LIN {X 0,Y 425.323,Z 412.747,A -85,B 0,C 180,E1 20527.293,E2 20527.293} C_VEL
LIN {X 0,Y 425.31,Z 412.73,A -85,B 0,C 180,E1 20523.37,E2 20523.37} C_VEL
LIN {X 0,Y 425.312,Z 412.748,A -85,B 0,C 180,E1 20519.596,E2 20519.596} C_VEL
LIN {X 0,Y 425.314,Z 412.756,A -85,B 0,C 180,E1 20515.686,E2 20515.686} C_VEL
LIN {X 0,Y 425.313,Z 412.739,A -85,B 0,C 180,E1 20511.785,E2 20511.785} C_VEL
LIN {X 0,Y 425.305,Z 412.739,A -85,B 0,C 180,E1 20507.923,E2 20507.923} C_VEL
LIN {X 0,Y 425.305,Z 412.745,A -85,B 0,C 180,E1 20504.035,E2 20504.035} C_VEL
LIN {X 0,Y 425.315,Z 412.752,A -85,B 0,C 180,E1 20500.213,E2 20500.213} C_VEL
LIN {X 0,Y 425.319,Z 412.753,A -85,B 0,C 180,E1 20496.445,E2 20496.445} C_VEL
LIN {X 0,Y 425.317,Z 412.751,A -85,B 0,C 180,E1 20492.564,E2 20492.564} C_VEL
LIN {X 0,Y 425.318,Z 412.746,A -85,B 0,C 180,E1 20488.699,E2 20488.699} C_VEL
LIN {X 0,Y 425.308,Z 412.744,A -85,B 0,C 180,E1 20484.833,E2 20484.833} C_VEL
LIN {X 0,Y 425.354,Z 413.101,A -85,B 0,C 180,E1 20483.004,E2 20483.004} C_VEL
LIN {X 0,Y 426.927,Z 416.653,A -85,B 0,C 180,E1 20482.32,E2 20482.32} C_VEL
LIN {X 0,Y 432.518,Z 427.517,A -85,B 0,C 180,E1 20480.338,E2 20480.338} C_VEL
LIN {X 0,Y 440.168,Z 443.004,A -85,B 0,C 180,E1 20477.75,E2 20477.75} C_VEL
LIN {X 0,Y 445.904,Z 455.372,A -85,B 0,C 180,E1 20475.919,E2 20475.919} C_VEL
LIN {X 0,Y 457.025,Z 473.943,A -85,B 0,C 180,E1 20474.241,E2 20474.241} C_VEL
LIN {X 0,Y 458.912,Z 489.017,A -85,B 0,C 180,E1 20473.725,E2 20473.725} C_VEL
LIN {X 0,Y 453.234,Z 708.899,A -85,B 0,C 180,E1 20469.92,E2 20469.92} C_VEL
LIN {X 0,Y 451.808,Z 759.725,A -85,B 0,C 180,E1 20469.018,E2 20469.018} C_VEL
LIN {X 0,Y 450.365,Z 781.628,A -85,B 0,C 180,E1 20468.419,E2 20468.419} C_VEL
LIN {X 0,Y 448.539,Z 802.923,A -85,B 0,C 180,E1 20467.608,E2 20467.608} C_VEL
LIN {X 0,Y 446.493,Z 822.784,A -85,B 0,C 180,E1 20466.642,E2 20466.642} C_VEL
LIN {X 0,Y 444.028,Z 843.126,A -85,B 0,C 180,E1 20465.399,E2 20465.399} C_VEL
LIN {X 0,Y 441.405,Z 862.685,A -85,B 0,C 180,E1 20463.945,E2 20463.945} C_VEL
LIN {X 0,Y 438.705,Z 881.613,A -85,B 0,C 180,E1 20462.27,E2 20462.27} C_VEL
LIN {X 0,Y 436.022,Z 899.637,A -85,B 0,C 180,E1 20460.376,E2 20460.376} C_VEL
LIN {X 0,Y 433.447,Z 916.409,A -85,B 0,C 180,E1 20458.299,E2 20458.299} C_VEL
LIN {X 0,Y 430.956,Z 933.189,A -85,B 0,C 180,E1 20455.863,E2 20455.863} C_VEL
LIN {X 0,Y 429.001,Z 947.176,A -85,B 0,C 180,E1 20453.489,E2 20453.489} C_VEL
LIN {X 0,Y 427.354,Z 959.751,A -85,B 0,C 180,E1 20450.978,E2 20450.978} C_VEL
LIN {X 0,Y 426.064,Z 971.018,A -85,B 0,C 180,E1 20448.331,E2 20448.331} C_VEL
LIN {X 0,Y 425.116,Z 980.962,A -85,B 0,C 180,E1 20445.555,E2 20445.555} C_VEL
LIN {X 0,Y 424.496,Z 988.98,A -85,B 0,C 180,E1 20442.794,E2 20442.794} C_VEL
LIN {X 0,Y 424.128,Z 995.597,A -85,B 0,C 180,E1 20439.912,E2 20439.912} C_VEL
LIN {X 0,Y 423.966,Z 1000.343,A -85,B 0,C 180,E1 20437.183,E2 20437.183} C_VEL
LIN {X 0,Y 423.919,Z 1003.442,A -85,B 0,C 180,E1 20434.467,E2 20434.467} C_VEL
LIN {X 0,Y 423.901,Z 1005.174,A -85,B 0,C 180,E1 20431.76,E2 20431.76} C_VEL
LIN {X 0,Y 423.901,Z 1005.321,A -85,B 0,C 180,E1 20429.057,E2 20429.057} C_VEL
LIN {X 0,Y 423.913,Z 1004.043,A -85,B 0,C 180,E1 20426.216,E2 20426.216} C_VEL
LIN {X 0,Y 423.96,Z 1001.217,A -85,B 0,C 180,E1 20423.503,E2 20423.503} C_VEL
LIN {X 0,Y 424.094,Z 996.661,A -85,B 0,C 180,E1 20420.641,E2 20420.641} C_VEL
LIN {X 0,Y 424.374,Z 991.039,A -85,B 0,C 180,E1 20418.037,E2 20418.037} C_VEL
LIN {X 0,Y 424.881,Z 983.447,A -85,B 0,C 180,E1 20415.28,E2 20415.28} C_VEL
LIN {X 0,Y 425.72,Z 974.127,A -85,B 0,C 180,E1 20412.508,E2 20412.508} C_VEL
LIN {X 0,Y 426.887,Z 963.337,A -85,B 0,C 180,E1 20409.864,E2 20409.864} C_VEL
LIN {X 0,Y 428.486,Z 950.359,A -85,B 0,C 180,E1 20407.178,E2 20407.178} C_VEL
LIN {X 0,Y 430.41,Z 936.295,A -85,B 0,C 180,E1 20404.699,E2 20404.699} C_VEL
LIN {X 0,Y 432.667,Z 920.798,A -85,B 0,C 180,E1 20402.368,E2 20402.368} C_VEL
LIN {X 0,Y 435.099,Z 904.208,A -85,B 0,C 180,E1 20400.244,E2 20400.244} C_VEL
LIN {X 0,Y 437.815,Z 885.884,A -85,B 0,C 180,E1 20398.242,E2 20398.242} C_VEL
LIN {X 0,Y 440.47,Z 867.438,A -85,B 0,C 180,E1 20396.527,E2 20396.527} C_VEL
LIN {X 0,Y 443.06,Z 848.116,A -85,B 0,C 180,E1 20395.031,E2 20395.031} C_VEL
LIN {X 0,Y 445.48,Z 828.163,A -85,B 0,C 180,E1 20393.747,E2 20393.747} C_VEL
LIN {X 0,Y 447.727,Z 807.657,A -85,B 0,C 180,E1 20392.674,E2 20392.674} C_VEL
LIN {X 0,Y 449.569,Z 787.136,A -85,B 0,C 180,E1 20391.839,E2 20391.839} C_VEL
LIN {X 0,Y 451.131,Z 764.896,A -85,B 0,C 180,E1 20391.175,E2 20391.175} C_VEL
LIN {X 0,Y 452.115,Z 740.735,A -85,B 0,C 180,E1 20390.686,E2 20390.686} C_VEL
LIN {X 0,Y 457.722,Z 517.41,A -85,B 0,C 180,E1 20386.836,E2 20386.836} C_VEL
LIN {X 0,Y 458.387,Z 486.605,A -85,B 0,C 180,E1 20386.272,E2 20386.272} C_VEL
LIN {X 0,Y 456.382,Z 472.949,A -85,B 0,C 180,E1 20385.758,E2 20385.758} C_VEL
LIN {X 0,Y 445.388,Z 454.22,A -85,B 0,C 180,E1 20384.011,E2 20384.011} C_VEL
LIN {X 0,Y 438.051,Z 438.21,A -85,B 0,C 180,E1 20381.447,E2 20381.447} C_VEL
LIN {X 0,Y 431.895,Z 425.933,A -85,B 0,C 180,E1 20379.198,E2 20379.198} C_VEL
LIN {X 0,Y 429.067,Z 420.711,A -85,B 0,C 180,E1 20378.136,E2 20378.136} C_VEL
LIN {X 0,Y 427.444,Z 417.332,A -85,B 0,C 180,E1 20377.458,E2 20377.458} C_VEL
LIN {X 0,Y 425.676,Z 414.437,A -85,B 0,C 180,E1 20376.785,E2 20376.785} C_VEL
LIN {X 0,Y 425.321,Z 412.922,A -85,B 0,C 180,E1 20376.4,E2 20376.4} C_VEL
LIN {X 0,Y 425.274,Z 412.761,A -85,B 0,C 180,E1 20372.689,E2 20372.689} C_VEL
LIN {X 0,Y 425.267,Z 412.756,A -85,B 0,C 180,E1 20368.968,E2 20368.968} C_VEL
LIN {X 0,Y 425.272,Z 412.763,A -85,B 0,C 180,E1 20365.185,E2 20365.185} C_VEL
LIN {X 0,Y 425.292,Z 412.751,A -85,B 0,C 180,E1 20361.422,E2 20361.422} C_VEL
LIN {X 0,Y 425.293,Z 412.749,A -85,B 0,C 180,E1 20357.654,E2 20357.654} C_VEL
LIN {X 0,Y 425.262,Z 412.756,A -85,B 0,C 180,E1 20353.875,E2 20353.875} C_VEL
LIN {X 0,Y 425.248,Z 412.764,A -85,B 0,C 180,E1 20350.156,E2 20350.156} C_VEL
LIN {X 0,Y 425.253,Z 412.763,A -85,B 0,C 180,E1 20346.344,E2 20346.344} C_VEL
LIN {X 0,Y 425.267,Z 412.754,A -85,B 0,C 180,E1 20342.56,E2 20342.56} C_VEL
LIN {X 0,Y 425.307,Z 412.749,A -85,B 0,C 180,E1 20338.922,E2 20338.922} C_VEL
LIN {X 0,Y 425.316,Z 412.758,A -85,B 0,C 180,E1 20335.01,E2 20335.01} C_VEL
LIN {X 0,Y 425.309,Z 412.75,A -85,B 0,C 180,E1 20331.21,E2 20331.21} C_VEL
LIN {X 0,Y 425.298,Z 412.76,A -85,B 0,C 180,E1 20327.37,E2 20327.37} C_VEL
LIN {X 0,Y 425.335,Z 413.097,A -85,B 0,C 180,E1 20325.767,E2 20325.767} C_VEL
LIN {X 0,Y 426.924,Z 416.643,A -85,B 0,C 180,E1 20324.932,E2 20324.932} C_VEL
LIN {X 0,Y 428.049,Z 418.942,A -85,B 0,C 180,E1 20324.417,E2 20324.417} C_VEL
LIN {X 0,Y 431.92,Z 426.469,A -85,B 0,C 180,E1 20322.764,E2 20322.764} C_VEL
LIN {X 0,Y 438.754,Z 441.345,A -85,B 0,C 180,E1 20319.872,E2 20319.872} C_VEL
LIN {X 0,Y 443.854,Z 453.504,A -85,B 0,C 180,E1 20317.803,E2 20317.803} C_VEL
LIN {X 0,Y 453.373,Z 469.49,A -85,B 0,C 180,E1 20316.249,E2 20316.249} C_VEL
LIN {X 0,Y 455.989,Z 486.254,A -85,B 0,C 180,E1 20315.571,E2 20315.571} C_VEL
LIN {X 0,Y 448.514,Z 720.49,A -85,B 0,C 180,E1 20311.323,E2 20311.323} C_VEL
LIN {X 0,Y 447.258,Z 741.418,A -85,B 0,C 180,E1 20310.709,E2 20310.709} C_VEL
LIN {X 0,Y 445.663,Z 761.022,A -85,B 0,C 180,E1 20309.905,E2 20309.905} C_VEL
LIN {X 0,Y 443.641,Z 781.159,A -85,B 0,C 180,E1 20308.827,E2 20308.827} C_VEL
LIN {X 0,Y 441.338,Z 800.443,A -85,B 0,C 180,E1 20307.525,E2 20307.525} C_VEL
LIN {X 0,Y 439.005,Z 817.909,A -85,B 0,C 180,E1 20306.082,E2 20306.082} C_VEL
LIN {X 0,Y 436.526,Z 834.898,A -85,B 0,C 180,E1 20304.395,E2 20304.395} C_VEL
LIN {X 0,Y 434.09,Z 850.626,A -85,B 0,C 180,E1 20302.518,E2 20302.518} C_VEL
LIN {X 0,Y 431.874,Z 864.692,A -85,B 0,C 180,E1 20300.526,E2 20300.526} C_VEL
LIN {X 0,Y 429.743,Z 878.309,A -85,B 0,C 180,E1 20298.241,E2 20298.241} C_VEL
LIN {X 0,Y 427.962,Z 890.347,A -85,B 0,C 180,E1 20295.822,E2 20295.822} C_VEL
LIN {X 0,Y 427.652,Z 892.536,A -85,B 0,C 180,E1 20295.33,E2 20295.33} C_VEL
LIN {X 0,Y 426.167,Z 896.521,A -85,B 0,C 180,E1 20294.457,E2 20294.457} C_VEL
LIN {X 0,Y 419.171,Z 906.089,A -85,B 0,C 180,E1 20292.243,E2 20292.243} C_VEL
LIN {X 0,Y 417.819,Z 909.262,A -85,B 0,C 180,E1 20291.294,E2 20291.294} C_VEL
LIN {X 0,Y 416.994,Z 916.645,A -85,B 0,C 180,E1 20288.561,E2 20288.561} C_VEL
LIN {X 0,Y 416.502,Z 922.575,A -85,B 0,C 180,E1 20285.681,E2 20285.681} C_VEL
LIN {X 0,Y 416.242,Z 926.666,A -85,B 0,C 180,E1 20282.875,E2 20282.875} C_VEL
LIN {X 0,Y 416.14,Z 929.15,A -85,B 0,C 180,E1 20280.12,E2 20280.12} C_VEL
LIN {X 0,Y 416.102,Z 930.046,A -85,B 0,C 180,E1 20277.316,E2 20277.316} C_VEL
LIN {X 0,Y 416.121,Z 929.428,A -85,B 0,C 180,E1 20274.558,E2 20274.558} C_VEL
LIN {X 0,Y 416.189,Z 927.235,A -85,B 0,C 180,E1 20271.71,E2 20271.71} C_VEL
LIN {X 0,Y 416.393,Z 923.475,A -85,B 0,C 180,E1 20268.898,E2 20268.898} C_VEL
LIN {X 0,Y 416.81,Z 917.853,A -85,B 0,C 180,E1 20266.01,E2 20266.01} C_VEL
LIN {X 0,Y 417.514,Z 910.766,A -85,B 0,C 180,E1 20263.288,E2 20263.288} C_VEL
LIN {X 0,Y 418.568,Z 901.959,A -85,B 0,C 180,E1 20260.596,E2 20260.596} C_VEL
LIN {X 0,Y 420.068,Z 891.24,A -85,B 0,C 180,E1 20257.932,E2 20257.932} C_VEL
LIN {X 0,Y 421.928,Z 879.061,A -85,B 0,C 180,E1 20255.436,E2 20255.436} C_VEL
LIN {X 0,Y 423.992,Z 866.293,A -85,B 0,C 180,E1 20253.242,E2 20253.242} C_VEL
LIN {X 0,Y 426.425,Z 851.282,A -85,B 0,C 180,E1 20251.072,E2 20251.072} C_VEL
LIN {X 0,Y 428.994,Z 835.029,A -85,B 0,C 180,E1 20249.113,E2 20249.113} C_VEL
LIN {X 0,Y 431.535,Z 818.021,A -85,B 0,C 180,E1 20247.408,E2 20247.408} C_VEL
LIN {X 0,Y 434.013,Z 799.936,A -85,B 0,C 180,E1 20245.902,E2 20245.902} C_VEL
LIN {X 0,Y 436.349,Z 780.844,A -85,B 0,C 180,E1 20244.607,E2 20244.607} C_VEL
LIN {X 0,Y 438.366,Z 761.267,A -85,B 0,C 180,E1 20243.548,E2 20243.548} C_VEL
LIN {X 0,Y 440.067,Z 740.96,A -85,B 0,C 180,E1 20242.708,E2 20242.708} C_VEL
LIN {X 0,Y 441.337,Z 720.076,A -85,B 0,C 180,E1 20242.095,E2 20242.095} C_VEL
LIN {X 0,Y 443.49,Z 649.085,A -85,B 0,C 180,E1 20240.797,E2 20240.797} C_VEL
LIN {X 0,Y 448.301,Z 485.674,A -85,B 0,C 180,E1 20237.865,E2 20237.865} C_VEL
LIN {X 0,Y 445.661,Z 471.282,A -85,B 0,C 180,E1 20237.262,E2 20237.262} C_VEL
LIN {X 0,Y 434.574,Z 452.493,A -85,B 0,C 180,E1 20235.506,E2 20235.506} C_VEL
LIN {X 0,Y 427.676,Z 436.344,A -85,B 0,C 180,E1 20232.725,E2 20232.725} C_VEL
LIN {X 0,Y 421.23,Z 422.181,A -85,B 0,C 180,E1 20230.048,E2 20230.048} C_VEL
LIN {X 0,Y 417.441,Z 414.135,A -85,B 0,C 180,E1 20228.385,E2 20228.385} C_VEL
LIN {X 0,Y 417.364,Z 413.685,A -85,B 0,C 180,E1 20227.459,E2 20227.459} C_VEL
LIN {X 0,Y 417.366,Z 413.742,A -85,B 0,C 180,E1 20223.537,E2 20223.537} C_VEL
LIN {X 0,Y 417.364,Z 413.734,A -85,B 0,C 180,E1 20219.634,E2 20219.634} C_VEL
LIN {X 0,Y 417.368,Z 413.731,A -85,B 0,C 180,E1 20215.736,E2 20215.736} C_VEL
LIN {X 0,Y 417.38,Z 413.729,A -85,B 0,C 180,E1 20211.79,E2 20211.79} C_VEL
LIN {X 0,Y 417.375,Z 413.736,A -85,B 0,C 180,E1 20207.872,E2 20207.872} C_VEL
LIN {X 0,Y 417.375,Z 413.744,A -85,B 0,C 180,E1 20204.006,E2 20204.006} C_VEL
LIN {X 0,Y 417.379,Z 413.738,A -85,B 0,C 180,E1 20200.122,E2 20200.122} C_VEL
LIN {X 0,Y 417.373,Z 413.723,A -85,B 0,C 180,E1 20196.279,E2 20196.279} C_VEL
LIN {X 0,Y 417.371,Z 413.733,A -85,B 0,C 180,E1 20192.454,E2 20192.454} C_VEL
LIN {X 0,Y 417.372,Z 413.745,A -85,B 0,C 180,E1 20188.628,E2 20188.628} C_VEL
LIN {X 0,Y 417.373,Z 413.725,A -85,B 0,C 180,E1 20184.776,E2 20184.776} C_VEL
LIN {X 0,Y 417.373,Z 413.724,A -85,B 0,C 180,E1 20180.884,E2 20180.884} C_VEL
LIN {X 0,Y 417.371,Z 413.746,A -85,B 0,C 180,E1 20176.994,E2 20176.994} C_VEL
LIN {X 0,Y 417.372,Z 413.733,A -85,B 0,C 180,E1 20173.155,E2 20173.155} C_VEL
LIN {X 0,Y 417.373,Z 413.723,A -85,B 0,C 180,E1 20169.237,E2 20169.237} C_VEL
LIN {X 0,Y 417.375,Z 413.74,A -85,B 0,C 180,E1 20165.361,E2 20165.361} C_VEL
LIN {X 0,Y 417.373,Z 413.738,A -85,B 0,C 180,E1 20161.51,E2 20161.51} C_VEL
LIN {X 0,Y 417.373,Z 413.723,A -85,B 0,C 180,E1 20157.666,E2 20157.666} C_VEL
LIN {X 0,Y 417.376,Z 413.729,A -85,B 0,C 180,E1 20153.812,E2 20153.812} C_VEL
LIN {X 0,Y 417.368,Z 413.748,A -85,B 0,C 180,E1 20149.929,E2 20149.929} C_VEL
LIN {X 0,Y 417.367,Z 413.743,A -85,B 0,C 180,E1 20145.99,E2 20145.99} C_VEL
LIN {X 0,Y 417.37,Z 413.738,A -85,B 0,C 180,E1 20142.144,E2 20142.144} C_VEL
LIN {X 0,Y 417.381,Z 413.732,A -85,B 0,C 180,E1 20138.204,E2 20138.204} C_VEL
LIN {X 0,Y 417.378,Z 413.734,A -85,B 0,C 180,E1 20134.258,E2 20134.258} C_VEL
LIN {X 0,Y 417.377,Z 413.738,A -85,B 0,C 180,E1 20130.414,E2 20130.414} C_VEL
LIN {X 0,Y 417.379,Z 413.748,A -85,B 0,C 180,E1 20126.479,E2 20126.479} C_VEL
LIN {X 0,Y 417.415,Z 414.005,A -85,B 0,C 180,E1 20124.199,E2 20124.199} C_VEL
LIN {X 0,Y 418.766,Z 417.366,A -85,B 0,C 180,E1 20123.522,E2 20123.522} C_VEL
LIN {X 0,Y 420.222,Z 420.029,A -85,B 0,C 180,E1 20122.989,E2 20122.989} C_VEL
LIN {X 0,Y 424.613,Z 428.405,A -85,B 0,C 180,E1 20121.391,E2 20121.391} C_VEL
LIN {X 0,Y 432.15,Z 443.536,A -85,B 0,C 180,E1 20118.746,E2 20118.746} C_VEL
LIN {X 0,Y 437.769,Z 455.416,A -85,B 0,C 180,E1 20116.906,E2 20116.906} C_VEL
LIN {X 0,Y 450.753,Z 476.655,A -85,B 0,C 180,E1 20114.893,E2 20114.893} C_VEL
LIN {X 0,Y 451.449,Z 478.644,A -85,B 0,C 180,E1 20114.771,E2 20114.771} C_VEL
LIN {X 0,Y 452.843,Z 490.465,A -85,B 0,C 180,E1 20114.365,E2 20114.365} C_VEL
LIN {X 0,Y 446.867,Z 708.641,A -85,B 0,C 180,E1 20110.543,E2 20110.543} C_VEL
LIN {X 0,Y 445.383,Z 759.282,A -85,B 0,C 180,E1 20109.635,E2 20109.635} C_VEL
LIN {X 0,Y 443.866,Z 781.223,A -85,B 0,C 180,E1 20109.032,E2 20109.032} C_VEL
LIN {X 0,Y 441.98,Z 802.261,A -85,B 0,C 180,E1 20108.225,E2 20108.225} C_VEL
LIN {X 0,Y 439.759,Z 822.742,A -85,B 0,C 180,E1 20107.216,E2 20107.216} C_VEL
LIN {X 0,Y 437.237,Z 842.472,A -85,B 0,C 180,E1 20105.996,E2 20105.996} C_VEL
LIN {X 0,Y 434.47,Z 862.048,A -85,B 0,C 180,E1 20104.526,E2 20104.526} C_VEL
LIN {X 0,Y 431.625,Z 881.014,A -85,B 0,C 180,E1 20102.826,E2 20102.826} C_VEL
LIN {X 0,Y 428.811,Z 898.807,A -85,B 0,C 180,E1 20100.934,E2 20100.934} C_VEL
LIN {X 0,Y 426.065,Z 915.747,A -85,B 0,C 180,E1 20098.808,E2 20098.808} C_VEL
LIN {X 0,Y 423.443,Z 932.379,A -85,B 0,C 180,E1 20096.356,E2 20096.356} C_VEL
LIN {X 0,Y 421.352,Z 946.392,A -85,B 0,C 180,E1 20093.942,E2 20093.942} C_VEL
LIN {X 0,Y 419.59,Z 958.978,A -85,B 0,C 180,E1 20091.385,E2 20091.385} C_VEL
LIN {X 0,Y 418.209,Z 970.266,A -85,B 0,C 180,E1 20088.688,E2 20088.688} C_VEL
LIN {X 0,Y 417.195,Z 980.224,A -85,B 0,C 180,E1 20085.858,E2 20085.858} C_VEL
LIN {X 0,Y 416.544,Z 988.249,A -85,B 0,C 180,E1 20083.043,E2 20083.043} C_VEL
LIN {X 0,Y 416.155,Z 994.879,A -85,B 0,C 180,E1 20080.104,E2 20080.104} C_VEL
LIN {X 0,Y 415.983,Z 999.627,A -85,B 0,C 180,E1 20077.322,E2 20077.322} C_VEL
LIN {X 0,Y 415.942,Z 1002.733,A -85,B 0,C 180,E1 20074.553,E2 20074.553} C_VEL
LIN {X 0,Y 415.93,Z 1004.48,A -85,B 0,C 180,E1 20071.794,E2 20071.794} C_VEL
LIN {X 0,Y 415.931,Z 1004.63,A -85,B 0,C 180,E1 20069.039,E2 20069.039} C_VEL
LIN {X 0,Y 415.939,Z 1003.439,A -85,B 0,C 180,E1 20066.282,E2 20066.282} C_VEL
LIN {X 0,Y 415.981,Z 1000.652,A -85,B 0,C 180,E1 20063.517,E2 20063.517} C_VEL
LIN {X 0,Y 416.106,Z 996.176,A -85,B 0,C 180,E1 20060.599,E2 20060.599} C_VEL
LIN {X 0,Y 416.389,Z 990.591,A -85,B 0,C 180,E1 20057.945,E2 20057.945} C_VEL
LIN {X 0,Y 416.952,Z 982.653,A -85,B 0,C 180,E1 20054.994,E2 20054.994} C_VEL
LIN {X 0,Y 417.808,Z 973.656,A -85,B 0,C 180,E1 20052.26,E2 20052.26} C_VEL
LIN {X 0,Y 419.084,Z 962.492,A -85,B 0,C 180,E1 20049.473,E2 20049.473} C_VEL
LIN {X 0,Y 420.768,Z 949.662,A -85,B 0,C 180,E1 20046.772,E2 20046.772} C_VEL
LIN {X 0,Y 422.766,Z 935.912,A -85,B 0,C 180,E1 20044.299,E2 20044.299} C_VEL
LIN {X 0,Y 425.137,Z 920.556,A -85,B 0,C 180,E1 20041.946,E2 20041.946} C_VEL
LIN {X 0,Y 427.661,Z 904.376,A -85,B 0,C 180,E1 20039.828,E2 20039.828} C_VEL
LIN {X 0,Y 430.511,Z 886.215,A -85,B 0,C 180,E1 20037.795,E2 20037.795} C_VEL
LIN {X 0,Y 433.301,Z 867.93,A -85,B 0,C 180,E1 20036.058,E2 20036.058} C_VEL
LIN {X 0,Y 436.016,Z 848.798,A -85,B 0,C 180,E1 20034.542,E2 20034.542} C_VEL
LIN {X 0,Y 438.772,Z 827.392,A -85,B 0,C 180,E1 20033.139,E2 20033.139} C_VEL
LIN {X 0,Y 441.18,Z 806.446,A -85,B 0,C 180,E1 20032.039,E2 20032.039} C_VEL
LIN {X 0,Y 443.091,Z 786.117,A -85,B 0,C 180,E1 20031.209,E2 20031.209} C_VEL
LIN {X 0,Y 444.694,Z 764.12,A -85,B 0,C 180,E1 20030.551,E2 20030.551} C_VEL
LIN {X 0,Y 445.739,Z 739.171,A -85,B 0,C 180,E1 20030.046,E2 20030.046} C_VEL
LIN {X 0,Y 451.718,Z 516.395,A -85,B 0,C 180,E1 20026.152,E2 20026.152} C_VEL
LIN {X 0,Y 452.376,Z 488.016,A -85,B 0,C 180,E1 20025.622,E2 20025.622} C_VEL
LIN {X 0,Y 450.777,Z 476.897,A -85,B 0,C 180,E1 20025.194,E2 20025.194} C_VEL
LIN {X 0,Y 439.621,Z 458.128,A -85,B 0,C 180,E1 20023.404,E2 20023.404} C_VEL
LIN {X 0,Y 437.261,Z 454.134,A -85,B 0,C 180,E1 20022.954,E2 20022.954} C_VEL
LIN {X 0,Y 430.662,Z 439.886,A -85,B 0,C 180,E1 20020.546,E2 20020.546} C_VEL
LIN {X 0,Y 424.742,Z 427.926,A -85,B 0,C 180,E1 20018.251,E2 20018.251} C_VEL
LIN {X 0,Y 421.603,Z 422.436,A -85,B 0,C 180,E1 20017.04,E2 20017.04} C_VEL
LIN {X 0,Y 419.365,Z 418.114,A -85,B 0,C 180,E1 20016.079,E2 20016.079} C_VEL
LIN {X 0,Y 417.515,Z 414.688,A -85,B 0,C 180,E1 20015.249,E2 20015.249} C_VEL
LIN {X 0,Y 417.349,Z 413.85,A -85,B 0,C 180,E1 20014.93,E2 20014.93} C_VEL
LIN {X 0,Y 417.331,Z 413.749,A -85,B 0,C 180,E1 20011.004,E2 20011.004} C_VEL
LIN {X 0,Y 417.335,Z 413.743,A -85,B 0,C 180,E1 20007.232,E2 20007.232} C_VEL
LIN {X 0,Y 417.352,Z 413.74,A -85,B 0,C 180,E1 20003.433,E2 20003.433} C_VEL
LIN {X 0,Y 417.357,Z 413.746,A -85,B 0,C 180,E1 19999.707,E2 19999.707} C_VEL
LIN {X 0,Y 417.333,Z 413.75,A -85,B 0,C 180,E1 19995.85,E2 19995.85} C_VEL
LIN {X 0,Y 417.307,Z 413.747,A -85,B 0,C 180,E1 19992.172,E2 19992.172} C_VEL
LIN {X 0,Y 417.31,Z 413.741,A -85,B 0,C 180,E1 19988.331,E2 19988.331} C_VEL
LIN {X 0,Y 417.322,Z 413.744,A -85,B 0,C 180,E1 19984.534,E2 19984.534} C_VEL
LIN {X 0,Y 417.354,Z 413.749,A -85,B 0,C 180,E1 19980.823,E2 19980.823} C_VEL
LIN {X 0,Y 417.371,Z 413.74,A -85,B 0,C 180,E1 19976.979,E2 19976.979} C_VEL
LIN {X 0,Y 417.379,Z 413.738,A -85,B 0,C 180,E1 19973.12,E2 19973.12} C_VEL
LIN {X 0,Y 417.368,Z 413.742,A -85,B 0,C 180,E1 19969.23,E2 19969.23} C_VEL
LIN {X 0,Y 417.406,Z 414.009,A -85,B 0,C 180,E1 19967.198,E2 19967.198} C_VEL
LIN {X 0,Y 418.833,Z 417.461,A -85,B 0,C 180,E1 19966.329,E2 19966.329} C_VEL
LIN {X 0,Y 420.011,Z 419.499,A -85,B 0,C 180,E1 19965.806,E2 19965.806} C_VEL
LIN {X 0,Y 422.515,Z 424.519,A -85,B 0,C 180,E1 19964.63,E2 19964.63} C_VEL
LIN {X 0,Y 426.558,Z 432.719,A -85,B 0,C 180,E1 19962.821,E2 19962.821} C_VEL
LIN {X 0,Y 432.441,Z 445.583,A -85,B 0,C 180,E1 19960.271,E2 19960.271} C_VEL
LIN {X 0,Y 435.951,Z 453.636,A -85,B 0,C 180,E1 19958.859,E2 19958.859} C_VEL
LIN {X 0,Y 446.554,Z 471.197,A -85,B 0,C 180,E1 19957.035,E2 19957.035} C_VEL
LIN {X 0,Y 447.991,Z 474.081,A -85,B 0,C 180,E1 19956.792,E2 19956.792} C_VEL
LIN {X 0,Y 450.046,Z 487.822,A -85,B 0,C 180,E1 19956.231,E2 19956.231} C_VEL
LIN {X 0,Y 442.145,Z 721.049,A -85,B 0,C 180,E1 19951.941,E2 19951.941} C_VEL
LIN {X 0,Y 440.822,Z 741.991,A -85,B 0,C 180,E1 19951.319,E2 19951.319} C_VEL
LIN {X 0,Y 439.127,Z 761.752,A -85,B 0,C 180,E1 19950.496,E2 19950.496} C_VEL
LIN {X 0,Y 437.033,Z 781.551,A -85,B 0,C 180,E1 19949.423,E2 19949.423} C_VEL
LIN {X 0,Y 434.673,Z 800.408,A -85,B 0,C 180,E1 19948.141,E2 19948.141} C_VEL
LIN {X 0,Y 432.239,Z 817.792,A -85,B 0,C 180,E1 19946.7,E2 19946.7} C_VEL
LIN {X 0,Y 429.612,Z 834.764,A -85,B 0,C 180,E1 19945,E2 19945} C_VEL
LIN {X 0,Y 427.011,Z 850.671,A -85,B 0,C 180,E1 19943.088,E2 19943.088} C_VEL
LIN {X 0,Y 424.557,Z 865.305,A -85,B 0,C 180,E1 19940.995,E2 19940.995} C_VEL
LIN {X 0,Y 422.253,Z 879.123,A -85,B 0,C 180,E1 19938.638,E2 19938.638} C_VEL
LIN {X 0,Y 420.357,Z 891.054,A -85,B 0,C 180,E1 19936.197,E2 19936.197} C_VEL
LIN {X 0,Y 418.855,Z 901.314,A -85,B 0,C 180,E1 19933.672,E2 19933.672} C_VEL
LIN {X 0,Y 417.819,Z 909.262,A -85,B 0,C 180,E1 19931.294,E2 19931.294} C_VEL
LIN {X 0,Y 416.505,Z 912.301,A -85,B 0,C 180,E1 19930.33,E2 19930.33} C_VEL
LIN {X 0,Y 409.629,Z 919.675,A -85,B 0,C 180,E1 19927.729,E2 19927.729} C_VEL
LIN {X 0,Y 408.726,Z 921.555,A -85,B 0,C 180,E1 19926.843,E2 19926.843} C_VEL
LIN {X 0,Y 408.378,Z 926.007,A -85,B 0,C 180,E1 19924.098,E2 19924.098} C_VEL
LIN {X 0,Y 408.209,Z 929.181,A -85,B 0,C 180,E1 19921.115,E2 19921.115} C_VEL
LIN {X 0,Y 408.142,Z 930.623,A -85,B 0,C 180,E1 19918.372,E2 19918.372} C_VEL
LIN {X 0,Y 408.137,Z 930.571,A -85,B 0,C 180,E1 19915.537,E2 19915.537} C_VEL
LIN {X 0,Y 408.194,Z 929.009,A -85,B 0,C 180,E1 19912.765,E2 19912.765} C_VEL
LIN {X 0,Y 408.349,Z 925.865,A -85,B 0,C 180,E1 19909.894,E2 19909.894} C_VEL
LIN {X 0,Y 408.681,Z 921.186,A -85,B 0,C 180,E1 19907.069,E2 19907.069} C_VEL
LIN {X 0,Y 409.293,Z 914.91,A -85,B 0,C 180,E1 19904.281,E2 19904.281} C_VEL
LIN {X 0,Y 410.253,Z 906.895,A -85,B 0,C 180,E1 19901.525,E2 19901.525} C_VEL
LIN {X 0,Y 411.561,Z 897.627,A -85,B 0,C 180,E1 19898.942,E2 19898.942} C_VEL
LIN {X 0,Y 413.411,Z 885.865,A -85,B 0,C 180,E1 19896.245,E2 19896.245} C_VEL
LIN {X 0,Y 415.517,Z 873.323,A -85,B 0,C 180,E1 19893.86,E2 19893.86} C_VEL
LIN {X 0,Y 417.911,Z 859.442,A -85,B 0,C 180,E1 19891.642,E2 19891.642} C_VEL
LIN {X 0,Y 420.515,Z 844.134,A -85,B 0,C 180,E1 19889.588,E2 19889.588} C_VEL
LIN {X 0,Y 423.168,Z 827.814,A -85,B 0,C 180,E1 19887.763,E2 19887.763} C_VEL
LIN {X 0,Y 425.757,Z 810.682,A -85,B 0,C 180,E1 19886.16,E2 19886.16} C_VEL
LIN {X 0,Y 428.365,Z 791.828,A -85,B 0,C 180,E1 19884.707,E2 19884.707} C_VEL
LIN {X 0,Y 430.626,Z 772.87,A -85,B 0,C 180,E1 19883.525,E2 19883.525} C_VEL
LIN {X 0,Y 432.625,Z 752.929,A -85,B 0,C 180,E1 19882.549,E2 19882.549} C_VEL
LIN {X 0,Y 434.213,Z 732.026,A -85,B 0,C 180,E1 19881.789,E2 19881.789} C_VEL
LIN {X 0,Y 435.274,Z 710.863,A -85,B 0,C 180,E1 19881.273,E2 19881.273} C_VEL
LIN {X 0,Y 442.296,Z 487.713,A -85,B 0,C 180,E1 19877.235,E2 19877.235} C_VEL
LIN {X 0,Y 440.084,Z 475.403,A -85,B 0,C 180,E1 19876.71,E2 19876.71} C_VEL
LIN {X 0,Y 428.455,Z 455.92,A -85,B 0,C 180,E1 19874.846,E2 19874.846} C_VEL
LIN {X 0,Y 426.291,Z 452.165,A -85,B 0,C 180,E1 19874.419,E2 19874.419} C_VEL
LIN {X 0,Y 419.176,Z 435.572,A -85,B 0,C 180,E1 19871.429,E2 19871.429} C_VEL
LIN {X 0,Y 412.902,Z 422.514,A -85,B 0,C 180,E1 19868.796,E2 19868.796} C_VEL
LIN {X 0,Y 410.993,Z 418.548,A -85,B 0,C 180,E1 19867.957,E2 19867.957} C_VEL
LIN {X 0,Y 409.469,Z 414.9,A -85,B 0,C 180,E1 19867.138,E2 19867.138} C_VEL
LIN {X 0,Y 409.434,Z 414.726,A -85,B 0,C 180,E1 19863.296,E2 19863.296} C_VEL
LIN {X 0,Y 409.427,Z 414.72,A -85,B 0,C 180,E1 19859.47,E2 19859.47} C_VEL
LIN {X 0,Y 409.427,Z 414.718,A -85,B 0,C 180,E1 19855.632,E2 19855.632} C_VEL
LIN {X 0,Y 409.435,Z 414.717,A -85,B 0,C 180,E1 19851.661,E2 19851.661} C_VEL
LIN {X 0,Y 409.436,Z 414.722,A -85,B 0,C 180,E1 19847.727,E2 19847.727} C_VEL
LIN {X 0,Y 409.439,Z 414.732,A -85,B 0,C 180,E1 19843.717,E2 19843.717} C_VEL
LIN {X 0,Y 409.439,Z 414.73,A -85,B 0,C 180,E1 19839.712,E2 19839.712} C_VEL
LIN {X 0,Y 409.433,Z 414.716,A -85,B 0,C 180,E1 19835.708,E2 19835.708} C_VEL
LIN {X 0,Y 409.435,Z 414.713,A -85,B 0,C 180,E1 19831.804,E2 19831.804} C_VEL
LIN {X 0,Y 409.444,Z 414.73,A -85,B 0,C 180,E1 19827.868,E2 19827.868} C_VEL
LIN {X 0,Y 409.437,Z 414.728,A -85,B 0,C 180,E1 19823.915,E2 19823.915} C_VEL
LIN {X 0,Y 409.432,Z 414.708,A -85,B 0,C 180,E1 19819.992,E2 19819.992} C_VEL
LIN {X 0,Y 409.431,Z 414.724,A -85,B 0,C 180,E1 19816.019,E2 19816.019} C_VEL
LIN {X 0,Y 409.435,Z 414.734,A -85,B 0,C 180,E1 19812.124,E2 19812.124} C_VEL
LIN {X 0,Y 409.436,Z 414.711,A -85,B 0,C 180,E1 19808.143,E2 19808.143} C_VEL
LIN {X 0,Y 409.431,Z 414.716,A -85,B 0,C 180,E1 19804.342,E2 19804.342} C_VEL
LIN {X 0,Y 409.43,Z 414.733,A -85,B 0,C 180,E1 19800.42,E2 19800.42} C_VEL
LIN {X 0,Y 409.429,Z 414.724,A -85,B 0,C 180,E1 19796.5,E2 19796.5} C_VEL
LIN {X 0,Y 409.434,Z 414.709,A -85,B 0,C 180,E1 19792.521,E2 19792.521} C_VEL
LIN {X 0,Y 409.435,Z 414.718,A -85,B 0,C 180,E1 19788.592,E2 19788.592} C_VEL
LIN {X 0,Y 409.438,Z 414.729,A -85,B 0,C 180,E1 19784.708,E2 19784.708} C_VEL
LIN {X 0,Y 409.439,Z 414.732,A -85,B 0,C 180,E1 19780.751,E2 19780.751} C_VEL
LIN {X 0,Y 409.441,Z 414.734,A -85,B 0,C 180,E1 19776.849,E2 19776.849} C_VEL
LIN {X 0,Y 409.441,Z 414.732,A -85,B 0,C 180,E1 19772.829,E2 19772.829} C_VEL
LIN {X 0,Y 409.437,Z 414.726,A -85,B 0,C 180,E1 19768.985,E2 19768.985} C_VEL
LIN {X 0,Y 409.463,Z 414.986,A -85,B 0,C 180,E1 19765.432,E2 19765.432} C_VEL
LIN {X 0,Y 410.704,Z 418.154,A -85,B 0,C 180,E1 19764.762,E2 19764.762} C_VEL
LIN {X 0,Y 411.874,Z 419.829,A -85,B 0,C 180,E1 19764.365,E2 19764.365} C_VEL
LIN {X 0,Y 418.977,Z 433.76,A -85,B 0,C 180,E1 19761.65,E2 19761.65} C_VEL
LIN {X 0,Y 426.83,Z 449.76,A -85,B 0,C 180,E1 19758.834,E2 19758.834} C_VEL
LIN {X 0,Y 429.591,Z 455.433,A -85,B 0,C 180,E1 19757.954,E2 19757.954} C_VEL
LIN {X 0,Y 443.519,Z 477.862,A -85,B 0,C 180,E1 19755.71,E2 19755.71} C_VEL
LIN {X 0,Y 445.732,Z 482.102,A -85,B 0,C 180,E1 19755.358,E2 19755.358} C_VEL
LIN {X 0,Y 446.822,Z 491.889,A -85,B 0,C 180,E1 19755.02,E2 19755.02} C_VEL
LIN {X 0,Y 440.501,Z 710.052,A -85,B 0,C 180,E1 19751.153,E2 19751.153} C_VEL
LIN {X 0,Y 438.983,Z 758.957,A -85,B 0,C 180,E1 19750.264,E2 19750.264} C_VEL
LIN {X 0,Y 437.383,Z 780.999,A -85,B 0,C 180,E1 19749.653,E2 19749.653} C_VEL
LIN {X 0,Y 435.385,Z 802.245,A -85,B 0,C 180,E1 19748.827,E2 19748.827} C_VEL
LIN {X 0,Y 433.066,Z 822.65,A -85,B 0,C 180,E1 19747.808,E2 19747.808} C_VEL
LIN {X 0,Y 430.426,Z 842.366,A -85,B 0,C 180,E1 19746.575,E2 19746.575} C_VEL
LIN {X 0,Y 427.572,Z 861.479,A -85,B 0,C 180,E1 19745.12,E2 19745.12} C_VEL
LIN {X 0,Y 424.648,Z 880.073,A -85,B 0,C 180,E1 19743.436,E2 19743.436} C_VEL
LIN {X 0,Y 421.669,Z 897.756,A -85,B 0,C 180,E1 19741.535,E2 19741.535} C_VEL
LIN {X 0,Y 418.878,Z 914.187,A -85,B 0,C 180,E1 19739.456,E2 19739.456} C_VEL
LIN {X 0,Y 416.258,Z 929.816,A -85,B 0,C 180,E1 19737.156,E2 19737.156} C_VEL
LIN {X 0,Y 413.954,Z 944.04,A -85,B 0,C 180,E1 19734.702,E2 19734.702} C_VEL
LIN {X 0,Y 412.025,Z 956.881,A -85,B 0,C 180,E1 19732.097,E2 19732.097} C_VEL
LIN {X 0,Y 410.431,Z 968.973,A -85,B 0,C 180,E1 19729.203,E2 19729.203} C_VEL
LIN {X 0,Y 409.328,Z 979.051,A -85,B 0,C 180,E1 19726.317,E2 19726.317} C_VEL
LIN {X 0,Y 408.618,Z 987.15,A -85,B 0,C 180,E1 19723.444,E2 19723.444} C_VEL
LIN {X 0,Y 408.206,Z 993.891,A -85,B 0,C 180,E1 19720.446,E2 19720.446} C_VEL
LIN {X 0,Y 408.017,Z 998.478,A -85,B 0,C 180,E1 19717.749,E2 19717.749} C_VEL
LIN {X 0,Y 407.961,Z 1001.901,A -85,B 0,C 180,E1 19714.783,E2 19714.783} C_VEL
LIN {X 0,Y 407.964,Z 1003.638,A -85,B 0,C 180,E1 19712.11,E2 19712.11} C_VEL
LIN {X 0,Y 407.956,Z 1003.962,A -85,B 0,C 180,E1 19709.301,E2 19709.301} C_VEL
LIN {X 0,Y 407.967,Z 1002.968,A -85,B 0,C 180,E1 19706.631,E2 19706.631} C_VEL
LIN {X 0,Y 407.998,Z 1000.255,A -85,B 0,C 180,E1 19703.672,E2 19703.672} C_VEL
LIN {X 0,Y 408.11,Z 995.959,A -85,B 0,C 180,E1 19700.698,E2 19700.698} C_VEL
LIN {X 0,Y 408.404,Z 990.144,A -85,B 0,C 180,E1 19697.849,E2 19697.849} C_VEL
LIN {X 0,Y 408.99,Z 982.288,A -85,B 0,C 180,E1 19694.84,E2 19694.84} C_VEL
LIN {X 0,Y 409.922,Z 973.02,A -85,B 0,C 180,E1 19691.958,E2 19691.958} C_VEL
LIN {X 0,Y 411.217,Z 962.252,A -85,B 0,C 180,E1 19689.211,E2 19689.211} C_VEL
LIN {X 0,Y 412.991,Z 949.517,A -85,B 0,C 180,E1 19686.459,E2 19686.459} C_VEL
LIN {X 0,Y 415.077,Z 935.991,A -85,B 0,C 180,E1 19683.961,E2 19683.961} C_VEL
LIN {X 0,Y 417.674,Z 920.044,A -85,B 0,C 180,E1 19681.467,E2 19681.467} C_VEL
LIN {X 0,Y 420.346,Z 903.966,A -85,B 0,C 180,E1 19679.326,E2 19679.326} C_VEL
LIN {X 0,Y 423.235,Z 886.553,A -85,B 0,C 180,E1 19677.334,E2 19677.334} C_VEL
LIN {X 0,Y 426.285,Z 867.632,A -85,B 0,C 180,E1 19675.502,E2 19675.502} C_VEL
LIN {X 0,Y 429.157,Z 848.483,A -85,B 0,C 180,E1 19673.962,E2 19673.962} C_VEL
LIN {X 0,Y 432.07,Z 827.021,A -85,B 0,C 180,E1 19672.536,E2 19672.536} C_VEL
LIN {X 0,Y 434.583,Z 806.325,A -85,B 0,C 180,E1 19671.433,E2 19671.433} C_VEL
LIN {X 0,Y 436.598,Z 785.953,A -85,B 0,C 180,E1 19670.59,E2 19670.59} C_VEL
LIN {X 0,Y 438.302,Z 763.85,A -85,B 0,C 180,E1 19669.919,E2 19669.919} C_VEL
LIN {X 0,Y 439.385,Z 739.646,A -85,B 0,C 180,E1 19669.42,E2 19669.42} C_VEL
LIN {X 0,Y 445.64,Z 520.31,A -85,B 0,C 180,E1 19665.538,E2 19665.538} C_VEL
LIN {X 0,Y 446.438,Z 489.488,A -85,B 0,C 180,E1 19664.956,E2 19664.956} C_VEL
LIN {X 0,Y 445.195,Z 480.762,A -85,B 0,C 180,E1 19664.612,E2 19664.612} C_VEL
LIN {X 0,Y 434.157,Z 462.176,A -85,B 0,C 180,E1 19662.772,E2 19662.772} C_VEL
LIN {X 0,Y 429.26,Z 454.242,A -85,B 0,C 180,E1 19661.861,E2 19661.861} C_VEL
LIN {X 0,Y 422.997,Z 441.044,A -85,B 0,C 180,E1 19659.482,E2 19659.482} C_VEL
LIN {X 0,Y 416.933,Z 429.026,A -85,B 0,C 180,E1 19657.008,E2 19657.008} C_VEL
LIN {X 0,Y 413.918,Z 423.671,A -85,B 0,C 180,E1 19655.751,E2 19655.751} C_VEL
LIN {X 0,Y 411.484,Z 419.212,A -85,B 0,C 180,E1 19654.652,E2 19654.652} C_VEL
LIN {X 0,Y 409.702,Z 416.01,A -85,B 0,C 180,E1 19653.808,E2 19653.808} C_VEL
LIN {X 0,Y 409.443,Z 414.939,A -85,B 0,C 180,E1 19653.496,E2 19653.496} C_VEL
LIN {X 0,Y 409.437,Z 414.727,A -85,B 0,C 180,E1 19649.718,E2 19649.718} C_VEL
LIN {X 0,Y 409.429,Z 414.73,A -85,B 0,C 180,E1 19645.765,E2 19645.765} C_VEL
LIN {X 0,Y 409.423,Z 414.731,A -85,B 0,C 180,E1 19641.789,E2 19641.789} C_VEL
LIN {X 0,Y 409.395,Z 414.729,A -85,B 0,C 180,E1 19637.922,E2 19637.922} C_VEL
LIN {X 0,Y 409.368,Z 414.732,A -85,B 0,C 180,E1 19634.137,E2 19634.137} C_VEL
LIN {X 0,Y 409.368,Z 414.742,A -85,B 0,C 180,E1 19630.27,E2 19630.27} C_VEL
LIN {X 0,Y 409.376,Z 414.742,A -85,B 0,C 180,E1 19626.31,E2 19626.31} C_VEL
LIN {X 0,Y 409.383,Z 414.73,A -85,B 0,C 180,E1 19622.379,E2 19622.379} C_VEL
LIN {X 0,Y 409.404,Z 414.73,A -85,B 0,C 180,E1 19618.6,E2 19618.6} C_VEL
LIN {X 0,Y 409.431,Z 414.737,A -85,B 0,C 180,E1 19614.815,E2 19614.815} C_VEL
LIN {X 0,Y 409.44,Z 414.726,A -85,B 0,C 180,E1 19611.008,E2 19611.008} C_VEL
LIN {X 0,Y 409.477,Z 415,A -85,B 0,C 180,E1 19608.735,E2 19608.735} C_VEL
LIN {X 0,Y 410.949,Z 418.552,A -85,B 0,C 180,E1 19607.779,E2 19607.779} C_VEL
LIN {X 0,Y 412.132,Z 420.36,A -85,B 0,C 180,E1 19607.245,E2 19607.245} C_VEL
LIN {X 0,Y 414.777,Z 425.708,A -85,B 0,C 180,E1 19605.908,E2 19605.908} C_VEL
LIN {X 0,Y 417.006,Z 430.107,A -85,B 0,C 180,E1 19604.849,E2 19604.849} C_VEL
LIN {X 0,Y 421.252,Z 438.937,A -85,B 0,C 180,E1 19602.883,E2 19602.883} C_VEL
LIN {X 0,Y 426.758,Z 451.133,A -85,B 0,C 180,E1 19600.425,E2 19600.425} C_VEL
LIN {X 0,Y 428.064,Z 453.927,A -85,B 0,C 180,E1 19599.971,E2 19599.971} C_VEL
LIN {X 0,Y 438.774,Z 471.232,A -85,B 0,C 180,E1 19598.039,E2 19598.039} C_VEL
LIN {X 0,Y 442.587,Z 478.227,A -85,B 0,C 180,E1 19597.371,E2 19597.371} C_VEL
LIN {X 0,Y 444.169,Z 489.431,A -85,B 0,C 180,E1 19596.909,E2 19596.909} C_VEL
LIN {X 0,Y 435.835,Z 721.494,A -85,B 0,C 180,E1 19592.581,E2 19592.581} C_VEL
LIN {X 0,Y 434.457,Z 742.405,A -85,B 0,C 180,E1 19591.952,E2 19591.952} C_VEL
LIN {X 0,Y 432.674,Z 762.231,A -85,B 0,C 180,E1 19591.12,E2 19591.12} C_VEL
LIN {X 0,Y 430.473,Z 782.1,A -85,B 0,C 180,E1 19590.03,E2 19590.03} C_VEL
LIN {X 0,Y 428.017,Z 800.741,A -85,B 0,C 180,E1 19588.75,E2 19588.75} C_VEL
LIN {X 0,Y 425.424,Z 818.291,A -85,B 0,C 180,E1 19587.278,E2 19587.278} C_VEL
LIN {X 0,Y 422.581,Z 835.745,A -85,B 0,C 180,E1 19585.505,E2 19585.505} C_VEL
LIN {X 0,Y 419.871,Z 851.388,A -85,B 0,C 180,E1 19583.593,E2 19583.593} C_VEL
LIN {X 0,Y 417.252,Z 866.054,A -85,B 0,C 180,E1 19581.461,E2 19581.461} C_VEL
LIN {X 0,Y 414.895,Z 879.314,A -85,B 0,C 180,E1 19579.169,E2 19579.169} C_VEL
LIN {X 0,Y 412.887,Z 891.112,A -85,B 0,C 180,E1 19576.739,E2 19576.739} C_VEL
LIN {X 0,Y 411.248,Z 901.477,A -85,B 0,C 180,E1 19574.173,E2 19574.173} C_VEL
LIN {X 0,Y 409.924,Z 910.873,A -85,B 0,C 180,E1 19571.3,E2 19571.3} C_VEL
LIN {X 0,Y 409.068,Z 917.983,A -85,B 0,C 180,E1 19568.541,E2 19568.541} C_VEL
LIN {X 0,Y 408.726,Z 921.555,A -85,B 0,C 180,E1 19566.843,E2 19566.843} C_VEL
LIN {X 0,Y 407.582,Z 923.608,A -85,B 0,C 180,E1 19565.805,E2 19565.805} C_VEL
LIN {X 0,Y 401.072,Z 928.187,A -85,B 0,C 180,E1 19563.004,E2 19563.004} C_VEL
LIN {X 0,Y 400.287,Z 929.221,A -85,B 0,C 180,E1 19562.066,E2 19562.066} C_VEL
LIN {X 0,Y 400.195,Z 931.078,A -85,B 0,C 180,E1 19559.152,E2 19559.152} C_VEL
LIN {X 0,Y 400.169,Z 931.408,A -85,B 0,C 180,E1 19556.233,E2 19556.233} C_VEL
LIN {X 0,Y 400.205,Z 930.277,A -85,B 0,C 180,E1 19553.402,E2 19553.402} C_VEL
LIN {X 0,Y 400.36,Z 927.521,A -85,B 0,C 180,E1 19550.461,E2 19550.461} C_VEL
LIN {X 0,Y 400.665,Z 923.157,A -85,B 0,C 180,E1 19547.571,E2 19547.571} C_VEL
LIN {X 0,Y 401.241,Z 917.241,A -85,B 0,C 180,E1 19544.721,E2 19544.721} C_VEL
LIN {X 0,Y 402.248,Z 909.235,A -85,B 0,C 180,E1 19541.757,E2 19541.757} C_VEL
LIN {X 0,Y 403.656,Z 899.797,A -85,B 0,C 180,E1 19538.974,E2 19538.974} C_VEL
LIN {X 0,Y 405.453,Z 889.026,A -85,B 0,C 180,E1 19536.368,E2 19536.368} C_VEL
LIN {X 0,Y 407.734,Z 876.154,A -85,B 0,C 180,E1 19533.793,E2 19533.793} C_VEL
LIN {X 0,Y 410.36,Z 861.668,A -85,B 0,C 180,E1 19531.393,E2 19531.393} C_VEL
LIN {X 0,Y 413.053,Z 846.56,A -85,B 0,C 180,E1 19529.304,E2 19529.304} C_VEL
LIN {X 0,Y 415.821,Z 830.573,A -85,B 0,C 180,E1 19527.448,E2 19527.448} C_VEL
LIN {X 0,Y 418.75,Z 812.321,A -85,B 0,C 180,E1 19525.683,E2 19525.683} C_VEL
LIN {X 0,Y 421.476,Z 793.718,A -85,B 0,C 180,E1 19524.211,E2 19524.211} C_VEL
LIN {X 0,Y 423.865,Z 774.903,A -85,B 0,C 180,E1 19523.001,E2 19523.001} C_VEL
LIN {X 0,Y 426.032,Z 754.407,A -85,B 0,C 180,E1 19521.97,E2 19521.97} C_VEL
LIN {X 0,Y 427.689,Z 733.766,A -85,B 0,C 180,E1 19521.202,E2 19521.202} C_VEL
LIN {X 0,Y 428.819,Z 713.039,A -85,B 0,C 180,E1 19520.671,E2 19520.671} C_VEL
LIN {X 0,Y 436.257,Z 489.229,A -85,B 0,C 180,E1 19516.567,E2 19516.567} C_VEL
LIN {X 0,Y 434.481,Z 479.354,A -85,B 0,C 180,E1 19516.133,E2 19516.133} C_VEL
LIN {X 0,Y 421.958,Z 458.349,A -85,B 0,C 180,E1 19514.054,E2 19514.054} C_VEL
LIN {X 0,Y 418.149,Z 452.119,A -85,B 0,C 180,E1 19513.323,E2 19513.323} C_VEL
LIN {X 0,Y 411.377,Z 436.611,A -85,B 0,C 180,E1 19510.4,E2 19510.4} C_VEL
LIN {X 0,Y 405.218,Z 423.866,A -85,B 0,C 180,E1 19507.714,E2 19507.714} C_VEL
LIN {X 0,Y 403.121,Z 419.607,A -85,B 0,C 180,E1 19506.771,E2 19506.771} C_VEL
LIN {X 0,Y 401.512,Z 415.886,A -85,B 0,C 180,E1 19505.893,E2 19505.893} C_VEL
LIN {X 0,Y 401.493,Z 415.711,A -85,B 0,C 180,E1 19501.919,E2 19501.919} C_VEL
LIN {X 0,Y 401.498,Z 415.712,A -85,B 0,C 180,E1 19497.963,E2 19497.963} C_VEL
LIN {X 0,Y 401.497,Z 415.712,A -85,B 0,C 180,E1 19494.002,E2 19494.002} C_VEL
LIN {X 0,Y 401.499,Z 415.707,A -85,B 0,C 180,E1 19490.019,E2 19490.019} C_VEL
LIN {X 0,Y 401.496,Z 415.701,A -85,B 0,C 180,E1 19485.986,E2 19485.986} C_VEL
LIN {X 0,Y 401.495,Z 415.701,A -85,B 0,C 180,E1 19482.06,E2 19482.06} C_VEL
LIN {X 0,Y 401.501,Z 415.713,A -85,B 0,C 180,E1 19478.097,E2 19478.097} C_VEL
LIN {X 0,Y 401.499,Z 415.722,A -85,B 0,C 180,E1 19474.079,E2 19474.079} C_VEL
LIN {X 0,Y 401.506,Z 415.708,A -85,B 0,C 180,E1 19470.036,E2 19470.036} C_VEL
LIN {X 0,Y 401.493,Z 415.695,A -85,B 0,C 180,E1 19466.155,E2 19466.155} C_VEL
LIN {X 0,Y 401.492,Z 415.717,A -85,B 0,C 180,E1 19462.243,E2 19462.243} C_VEL
LIN {X 0,Y 401.495,Z 415.715,A -85,B 0,C 180,E1 19458.288,E2 19458.288} C_VEL
LIN {X 0,Y 401.497,Z 415.697,A -85,B 0,C 180,E1 19454.273,E2 19454.273} C_VEL
LIN {X 0,Y 401.497,Z 415.711,A -85,B 0,C 180,E1 19450.33,E2 19450.33} C_VEL
LIN {X 0,Y 401.5,Z 415.721,A -85,B 0,C 180,E1 19446.291,E2 19446.291} C_VEL
LIN {X 0,Y 401.492,Z 415.701,A -85,B 0,C 180,E1 19442.284,E2 19442.284} C_VEL
LIN {X 0,Y 401.489,Z 415.701,A -85,B 0,C 180,E1 19438.431,E2 19438.431} C_VEL
LIN {X 0,Y 401.491,Z 415.719,A -85,B 0,C 180,E1 19434.427,E2 19434.427} C_VEL
LIN {X 0,Y 401.496,Z 415.722,A -85,B 0,C 180,E1 19430.468,E2 19430.468} C_VEL
LIN {X 0,Y 401.5,Z 415.715,A -85,B 0,C 180,E1 19426.462,E2 19426.462} C_VEL
LIN {X 0,Y 401.497,Z 415.708,A -85,B 0,C 180,E1 19422.463,E2 19422.463} C_VEL
LIN {X 0,Y 401.501,Z 415.705,A -85,B 0,C 180,E1 19418.527,E2 19418.527} C_VEL
LIN {X 0,Y 401.498,Z 415.707,A -85,B 0,C 180,E1 19414.638,E2 19414.638} C_VEL
LIN {X 0,Y 401.502,Z 415.71,A -85,B 0,C 180,E1 19410.648,E2 19410.648} C_VEL
LIN {X 0,Y 401.53,Z 415.946,A -85,B 0,C 180,E1 19406.761,E2 19406.761} C_VEL
LIN {X 0,Y 402.942,Z 419.398,A -85,B 0,C 180,E1 19405.977,E2 19405.977} C_VEL
LIN {X 0,Y 404.304,Z 421.74,A -85,B 0,C 180,E1 19405.441,E2 19405.441} C_VEL
LIN {X 0,Y 406.903,Z 426.735,A -85,B 0,C 180,E1 19404.383,E2 19404.383} C_VEL
LIN {X 0,Y 413.028,Z 438.313,A -85,B 0,C 180,E1 19402.057,E2 19402.057} C_VEL
LIN {X 0,Y 421.219,Z 455.149,A -85,B 0,C 180,E1 19399.092,E2 19399.092} C_VEL
LIN {X 0,Y 433.489,Z 474.523,A -85,B 0,C 180,E1 19397.011,E2 19397.011} C_VEL
LIN {X 0,Y 440.082,Z 485.935,A -85,B 0,C 180,E1 19395.943,E2 19395.943} C_VEL
LIN {X 0,Y 440.83,Z 493.461,A -85,B 0,C 180,E1 19395.687,E2 19395.687} C_VEL
LIN {X 0,Y 434.199,Z 710.93,A -85,B 0,C 180,E1 19391.791,E2 19391.791} C_VEL
LIN {X 0,Y 432.641,Z 758.585,A -85,B 0,C 180,E1 19390.913,E2 19390.913} C_VEL
LIN {X 0,Y 430.967,Z 780.638,A -85,B 0,C 180,E1 19390.296,E2 19390.296} C_VEL
LIN {X 0,Y 428.924,Z 801.367,A -85,B 0,C 180,E1 19389.486,E2 19389.486} C_VEL
LIN {X 0,Y 426.542,Z 821.613,A -85,B 0,C 180,E1 19388.471,E2 19388.471} C_VEL
LIN {X 0,Y 423.803,Z 841.142,A -85,B 0,C 180,E1 19387.242,E2 19387.242} C_VEL
LIN {X 0,Y 420.658,Z 861.247,A -85,B 0,C 180,E1 19385.701,E2 19385.701} C_VEL
LIN {X 0,Y 417.591,Z 879.815,A -85,B 0,C 180,E1 19383.995,E2 19383.995} C_VEL
LIN {X 0,Y 414.444,Z 897.537,A -85,B 0,C 180,E1 19382.059,E2 19382.059} C_VEL
LIN {X 0,Y 411.422,Z 914.369,A -85,B 0,C 180,E1 19379.883,E2 19379.883} C_VEL
LIN {X 0,Y 408.505,Z 930.741,A -85,B 0,C 180,E1 19377.399,E2 19377.399} C_VEL
LIN {X 0,Y 406.119,Z 944.819,A -85,B 0,C 180,E1 19374.9,E2 19374.9} C_VEL
LIN {X 0,Y 404.022,Z 958.089,A -85,B 0,C 180,E1 19372.099,E2 19372.099} C_VEL
LIN {X 0,Y 402.444,Z 969.466,A -85,B 0,C 180,E1 19369.25,E2 19369.25} C_VEL
LIN {X 0,Y 401.332,Z 979.174,A -85,B 0,C 180,E1 19366.354,E2 19366.354} C_VEL
LIN {X 0,Y 400.612,Z 987.16,A -85,B 0,C 180,E1 19363.424,E2 19363.424} C_VEL
LIN {X 0,Y 400.202,Z 993.71,A -85,B 0,C 180,E1 19360.366,E2 19360.366} C_VEL
LIN {X 0,Y 400.017,Z 998.4,A -85,B 0,C 180,E1 19357.471,E2 19357.471} C_VEL
LIN {X 0,Y 399.989,Z 1001.432,A -85,B 0,C 180,E1 19354.591,E2 19354.591} C_VEL
LIN {X 0,Y 399.992,Z 1003.088,A -85,B 0,C 180,E1 19351.722,E2 19351.722} C_VEL
LIN {X 0,Y 399.995,Z 1003.199,A -85,B 0,C 180,E1 19349,E2 19349} C_VEL
LIN {X 0,Y 399.995,Z 1001.989,A -85,B 0,C 180,E1 19346.133,E2 19346.133} C_VEL
LIN {X 0,Y 400.031,Z 999.181,A -85,B 0,C 180,E1 19343.257,E2 19343.257} C_VEL
LIN {X 0,Y 400.147,Z 994.666,A -85,B 0,C 180,E1 19340.221,E2 19340.221} C_VEL
LIN {X 0,Y 400.457,Z 989.051,A -85,B 0,C 180,E1 19337.458,E2 19337.458} C_VEL
LIN {X 0,Y 401.114,Z 981.065,A -85,B 0,C 180,E1 19334.386,E2 19334.386} C_VEL
LIN {X 0,Y 402.127,Z 971.658,A -85,B 0,C 180,E1 19331.446,E2 19331.446} C_VEL
LIN {X 0,Y 403.532,Z 960.802,A -85,B 0,C 180,E1 19328.644,E2 19328.644} C_VEL
LIN {X 0,Y 405.343,Z 948.644,A -85,B 0,C 180,E1 19325.987,E2 19325.987} C_VEL
LIN {X 0,Y 407.673,Z 934.433,A -85,B 0,C 180,E1 19323.336,E2 19323.336} C_VEL
LIN {X 0,Y 410.304,Z 919.165,A -85,B 0,C 180,E1 19320.916,E2 19320.916} C_VEL
LIN {X 0,Y 413.164,Z 902.996,A -85,B 0,C 180,E1 19318.733,E2 19318.733} C_VEL
LIN {X 0,Y 416.333,Z 884.844,A -85,B 0,C 180,E1 19316.64,E2 19316.64} C_VEL
LIN {X 0,Y 419.478,Z 866.393,A -85,B 0,C 180,E1 19314.841,E2 19314.841} C_VEL
LIN {X 0,Y 422.456,Z 847.438,A -85,B 0,C 180,E1 19313.306,E2 19313.306} C_VEL
LIN {X 0,Y 425.433,Z 826.677,A -85,B 0,C 180,E1 19311.913,E2 19311.913} C_VEL
LIN {X 0,Y 428.01,Z 806.581,A -85,B 0,C 180,E1 19310.823,E2 19310.823} C_VEL
LIN {X 0,Y 430.152,Z 785.944,A -85,B 0,C 180,E1 19309.957,E2 19309.957} C_VEL
LIN {X 0,Y 431.966,Z 763.593,A -85,B 0,C 180,E1 19309.268,E2 19309.268} C_VEL
LIN {X 0,Y 433.094,Z 739.833,A -85,B 0,C 180,E1 19308.77,E2 19308.77} C_VEL
LIN {X 0,Y 439.786,Z 519.325,A -85,B 0,C 180,E1 19304.815,E2 19304.815} C_VEL
LIN {X 0,Y 440.553,Z 490.872,A -85,B 0,C 180,E1 19304.269,E2 19304.269} C_VEL
LIN {X 0,Y 439.622,Z 484.695,A -85,B 0,C 180,E1 19304.012,E2 19304.012} C_VEL
LIN {X 0,Y 428.698,Z 466.045,A -85,B 0,C 180,E1 19302.108,E2 19302.108} C_VEL
LIN {X 0,Y 421.15,Z 454.226,A -85,B 0,C 180,E1 19300.669,E2 19300.669} C_VEL
LIN {X 0,Y 415.096,Z 441.762,A -85,B 0,C 180,E1 19298.246,E2 19298.246} C_VEL
LIN {X 0,Y 411.15,Z 434.072,A -85,B 0,C 180,E1 19296.57,E2 19296.57} C_VEL
LIN {X 0,Y 408.552,Z 429.252,A -85,B 0,C 180,E1 19295.424,E2 19295.424} C_VEL
LIN {X 0,Y 406.494,Z 425.317,A -85,B 0,C 180,E1 19294.453,E2 19294.453} C_VEL
LIN {X 0,Y 404.338,Z 421.153,A -85,B 0,C 180,E1 19293.381,E2 19293.381} C_VEL
LIN {X 0,Y 401.908,Z 417.483,A -85,B 0,C 180,E1 19292.246,E2 19292.246} C_VEL
LIN {X 0,Y 401.525,Z 415.921,A -85,B 0,C 180,E1 19291.783,E2 19291.783} C_VEL
LIN {X 0,Y 401.481,Z 415.727,A -85,B 0,C 180,E1 19288.079,E2 19288.079} C_VEL
LIN {X 0,Y 401.453,Z 415.72,A -85,B 0,C 180,E1 19284.264,E2 19284.264} C_VEL
LIN {X 0,Y 401.435,Z 415.72,A -85,B 0,C 180,E1 19280.54,E2 19280.54} C_VEL
LIN {X 0,Y 401.427,Z 415.73,A -85,B 0,C 180,E1 19276.644,E2 19276.644} C_VEL
LIN {X 0,Y 401.434,Z 415.731,A -85,B 0,C 180,E1 19272.807,E2 19272.807} C_VEL
LIN {X 0,Y 401.46,Z 415.719,A -85,B 0,C 180,E1 19269.027,E2 19269.027} C_VEL
LIN {X 0,Y 401.484,Z 415.713,A -85,B 0,C 180,E1 19265.287,E2 19265.287} C_VEL
LIN {X 0,Y 401.491,Z 415.717,A -85,B 0,C 180,E1 19261.284,E2 19261.284} C_VEL
LIN {X 0,Y 401.477,Z 415.726,A -85,B 0,C 180,E1 19257.43,E2 19257.43} C_VEL
LIN {X 0,Y 401.472,Z 415.717,A -85,B 0,C 180,E1 19253.523,E2 19253.523} C_VEL
LIN {X 0,Y 401.516,Z 415.961,A -85,B 0,C 180,E1 19250.468,E2 19250.468} C_VEL
LIN {X 0,Y 402.972,Z 419.473,A -85,B 0,C 180,E1 19249.42,E2 19249.42} C_VEL
LIN {X 0,Y 404.176,Z 421.064,A -85,B 0,C 180,E1 19248.874,E2 19248.874} C_VEL
LIN {X 0,Y 405.992,Z 424.817,A -85,B 0,C 180,E1 19247.858,E2 19247.858} C_VEL
LIN {X 0,Y 409.336,Z 431.314,A -85,B 0,C 180,E1 19246.15,E2 19246.15} C_VEL
LIN {X 0,Y 413.473,Z 439.671,A -85,B 0,C 180,E1 19244.141,E2 19244.141} C_VEL
LIN {X 0,Y 419.671,Z 453.277,A -85,B 0,C 180,E1 19241.274,E2 19241.274} C_VEL
LIN {X 0,Y 430.773,Z 470.846,A -85,B 0,C 180,E1 19239.145,E2 19239.145} C_VEL
LIN {X 0,Y 437.233,Z 482.252,A -85,B 0,C 180,E1 19237.973,E2 19237.973} C_VEL
LIN {X 0,Y 438.376,Z 491.059,A -85,B 0,C 180,E1 19237.608,E2 19237.608} C_VEL
LIN {X 0,Y 429.595,Z 722.034,A -85,B 0,C 180,E1 19233.24,E2 19233.24} C_VEL
LIN {X 0,Y 428.137,Z 743.081,A -85,B 0,C 180,E1 19232.598,E2 19232.598} C_VEL
LIN {X 0,Y 426.294,Z 762.551,A -85,B 0,C 180,E1 19231.77,E2 19231.77} C_VEL
LIN {X 0,Y 423.988,Z 782.453,A -85,B 0,C 180,E1 19230.669,E2 19230.669} C_VEL
LIN {X 0,Y 421.411,Z 801.151,A -85,B 0,C 180,E1 19229.373,E2 19229.373} C_VEL
LIN {X 0,Y 418.664,Z 818.821,A -85,B 0,C 180,E1 19227.875,E2 19227.875} C_VEL
LIN {X 0,Y 415.665,Z 836.279,A -85,B 0,C 180,E1 19226.078,E2 19226.078} C_VEL
LIN {X 0,Y 412.757,Z 852.141,A -85,B 0,C 180,E1 19224.11,E2 19224.11} C_VEL
LIN {X 0,Y 410,Z 866.692,A -85,B 0,C 180,E1 19221.963,E2 19221.963} C_VEL
LIN {X 0,Y 407.396,Z 880.492,A -85,B 0,C 180,E1 19219.53,E2 19219.53} C_VEL
LIN {X 0,Y 405.288,Z 892.079,A -85,B 0,C 180,E1 19217.085,E2 19217.085} C_VEL
LIN {X 0,Y 403.536,Z 902.402,A -85,B 0,C 180,E1 19214.472,E2 19214.472} C_VEL
LIN {X 0,Y 402.117,Z 911.766,A -85,B 0,C 180,E1 19211.545,E2 19211.545} C_VEL
LIN {X 0,Y 401.188,Z 918.871,A -85,B 0,C 180,E1 19208.717,E2 19208.717} C_VEL
LIN {X 0,Y 400.635,Z 924.454,A -85,B 0,C 180,E1 19205.796,E2 19205.796} C_VEL
LIN {X 0,Y 400.322,Z 928.443,A -85,B 0,C 180,E1 19202.814,E2 19202.814} C_VEL
LIN {X 0,Y 400.287,Z 929.221,A -85,B 0,C 180,E1 19202.066,E2 19202.066} C_VEL
LIN {X 0,Y 399.265,Z 930.273,A -85,B 0,C 180,E1 19200.974,E2 19200.974} C_VEL
LIN {X 0,Y 394.583,Z 931.717,A -85,B 0,C 180,E1 19198.907,E2 19198.907} C_VEL
LIN {X 0,Y 392.401,Z 932.167,A -85,B 0,C 180,E1 19197.557,E2 19197.557} C_VEL
LIN {X 0,Y 392.202,Z 932.234,A -85,B 0,C 180,E1 19197.068,E2 19197.068} C_VEL
LIN {X 0,Y 392.225,Z 931.403,A -85,B 0,C 180,E1 19194.067,E2 19194.067} C_VEL
LIN {X 0,Y 392.345,Z 928.995,A -85,B 0,C 180,E1 19191.055,E2 19191.055} C_VEL
LIN {X 0,Y 392.644,Z 925.053,A -85,B 0,C 180,E1 19188.096,E2 19188.096} C_VEL
LIN {X 0,Y 393.197,Z 919.574,A -85,B 0,C 180,E1 19185.18,E2 19185.18} C_VEL
LIN {X 0,Y 394.187,Z 912.005,A -85,B 0,C 180,E1 19182.15,E2 19182.15} C_VEL
LIN {X 0,Y 395.565,Z 902.978,A -85,B 0,C 180,E1 19179.306,E2 19179.306} C_VEL
LIN {X 0,Y 397.345,Z 892.639,A -85,B 0,C 180,E1 19176.644,E2 19176.644} C_VEL
LIN {X 0,Y 399.627,Z 880.311,A -85,B 0,C 180,E1 19174.014,E2 19174.014} C_VEL
LIN {X 0,Y 402.271,Z 866.491,A -85,B 0,C 180,E1 19171.564,E2 19171.564} C_VEL
LIN {X 0,Y 405.121,Z 851.636,A -85,B 0,C 180,E1 19169.361,E2 19169.361} C_VEL
LIN {X 0,Y 408.051,Z 835.88,A -85,B 0,C 180,E1 19167.399,E2 19167.399} C_VEL
LIN {X 0,Y 411.044,Z 818.5,A -85,B 0,C 180,E1 19165.603,E2 19165.603} C_VEL
LIN {X 0,Y 413.816,Z 800.943,A -85,B 0,C 180,E1 19164.103,E2 19164.103} C_VEL
LIN {X 0,Y 416.51,Z 781.654,A -85,B 0,C 180,E1 19162.757,E2 19162.757} C_VEL
LIN {X 0,Y 418.819,Z 761.832,A -85,B 0,C 180,E1 19161.658,E2 19161.658} C_VEL
LIN {X 0,Y 420.748,Z 741.519,A -85,B 0,C 180,E1 19160.801,E2 19160.801} C_VEL
LIN {X 0,Y 422.182,Z 720.594,A -85,B 0,C 180,E1 19160.171,E2 19160.171} C_VEL
LIN {X 0,Y 430.165,Z 495.125,A -85,B 0,C 180,E1 19155.966,E2 19155.966} C_VEL
LIN {X 0,Y 430.133,Z 489.81,A -85,B 0,C 180,E1 19155.84,E2 19155.84} C_VEL
LIN {X 0,Y 428.909,Z 483.379,A -85,B 0,C 180,E1 19155.541,E2 19155.541} C_VEL
LIN {X 0,Y 417.192,Z 463.603,A -85,B 0,C 180,E1 19153.535,E2 19153.535} C_VEL
LIN {X 0,Y 410.227,Z 452.563,A -85,B 0,C 180,E1 19152.259,E2 19152.259} C_VEL
LIN {X 0,Y 403.78,Z 438.061,A -85,B 0,C 180,E1 19149.395,E2 19149.395} C_VEL
LIN {X 0,Y 397.579,Z 425.235,A -85,B 0,C 180,E1 19146.585,E2 19146.585} C_VEL
LIN {X 0,Y 394.882,Z 420.193,A -85,B 0,C 180,E1 19145.369,E2 19145.369} C_VEL
LIN {X 0,Y 393.579,Z 416.845,A -85,B 0,C 180,E1 19144.527,E2 19144.527} C_VEL
LIN {X 0,Y 393.563,Z 416.714,A -85,B 0,C 180,E1 19140.623,E2 19140.623} C_VEL
LIN {X 0,Y 393.56,Z 416.707,A -85,B 0,C 180,E1 19136.541,E2 19136.541} C_VEL
LIN {X 0,Y 393.561,Z 416.71,A -85,B 0,C 180,E1 19132.611,E2 19132.611} C_VEL
LIN {X 0,Y 393.565,Z 416.71,A -85,B 0,C 180,E1 19128.657,E2 19128.657} C_VEL
LIN {X 0,Y 393.557,Z 416.709,A -85,B 0,C 180,E1 19124.652,E2 19124.652} C_VEL
LIN {X 0,Y 393.558,Z 416.697,A -85,B 0,C 180,E1 19120.566,E2 19120.566} C_VEL
LIN {X 0,Y 393.55,Z 416.687,A -85,B 0,C 180,E1 19116.596,E2 19116.596} C_VEL
LIN {X 0,Y 393.554,Z 416.699,A -85,B 0,C 180,E1 19112.589,E2 19112.589} C_VEL
LIN {X 0,Y 393.556,Z 416.711,A -85,B 0,C 180,E1 19108.531,E2 19108.531} C_VEL
LIN {X 0,Y 393.553,Z 416.694,A -85,B 0,C 180,E1 19104.464,E2 19104.464} C_VEL
LIN {X 0,Y 393.556,Z 416.684,A -85,B 0,C 180,E1 19100.524,E2 19100.524} C_VEL
LIN {X 0,Y 393.56,Z 416.706,A -85,B 0,C 180,E1 19096.532,E2 19096.532} C_VEL
LIN {X 0,Y 393.557,Z 416.703,A -85,B 0,C 180,E1 19092.621,E2 19092.621} C_VEL
LIN {X 0,Y 393.553,Z 416.685,A -85,B 0,C 180,E1 19088.621,E2 19088.621} C_VEL
LIN {X 0,Y 393.553,Z 416.698,A -85,B 0,C 180,E1 19084.664,E2 19084.664} C_VEL
LIN {X 0,Y 393.553,Z 416.71,A -85,B 0,C 180,E1 19080.583,E2 19080.583} C_VEL
LIN {X 0,Y 393.552,Z 416.698,A -85,B 0,C 180,E1 19076.651,E2 19076.651} C_VEL
LIN {X 0,Y 393.564,Z 416.684,A -85,B 0,C 180,E1 19072.703,E2 19072.703} C_VEL
LIN {X 0,Y 393.559,Z 416.695,A -85,B 0,C 180,E1 19068.718,E2 19068.718} C_VEL
LIN {X 0,Y 393.562,Z 416.706,A -85,B 0,C 180,E1 19064.68,E2 19064.68} C_VEL
LIN {X 0,Y 393.561,Z 416.71,A -85,B 0,C 180,E1 19060.715,E2 19060.715} C_VEL
LIN {X 0,Y 393.563,Z 416.71,A -85,B 0,C 180,E1 19056.652,E2 19056.652} C_VEL
LIN {X 0,Y 393.562,Z 416.706,A -85,B 0,C 180,E1 19052.624,E2 19052.624} C_VEL
LIN {X 0,Y 393.562,Z 416.698,A -85,B 0,C 180,E1 19048.611,E2 19048.611} C_VEL
LIN {X 0,Y 393.655,Z 417.283,A -85,B 0,C 180,E1 19048.015,E2 19048.015} C_VEL
LIN {X 0,Y 395.245,Z 420.722,A -85,B 0,C 180,E1 19047.224,E2 19047.224} C_VEL
LIN {X 0,Y 396.291,Z 422.449,A -85,B 0,C 180,E1 19046.805,E2 19046.805} C_VEL
LIN {X 0,Y 401.682,Z 432.769,A -85,B 0,C 180,E1 19044.551,E2 19044.551} C_VEL
LIN {X 0,Y 407.882,Z 444.814,A -85,B 0,C 180,E1 19042.126,E2 19042.126} C_VEL
LIN {X 0,Y 413.095,Z 455.28,A -85,B 0,C 180,E1 19040.239,E2 19040.239} C_VEL
LIN {X 0,Y 426.283,Z 475.732,A -85,B 0,C 180,E1 19037.915,E2 19037.915} C_VEL
LIN {X 0,Y 434.468,Z 489.724,A -85,B 0,C 180,E1 19036.543,E2 19036.543} C_VEL
LIN {X 0,Y 434.892,Z 495.038,A -85,B 0,C 180,E1 19036.371,E2 19036.371} C_VEL
LIN {X 0,Y 427.919,Z 712.249,A -85,B 0,C 180,E1 19032.435,E2 19032.435} C_VEL
LIN {X 0,Y 426.332,Z 758.36,A -85,B 0,C 180,E1 19031.574,E2 19031.574} C_VEL
LIN {X 0,Y 424.585,Z 780.477,A -85,B 0,C 180,E1 19030.951,E2 19030.951} C_VEL
LIN {X 0,Y 422.473,Z 800.95,A -85,B 0,C 180,E1 19030.144,E2 19030.144} C_VEL
LIN {X 0,Y 419.887,Z 821.854,A -85,B 0,C 180,E1 19029.079,E2 19029.079} C_VEL
LIN {X 0,Y 416.918,Z 842.072,A -85,B 0,C 180,E1 19027.783,E2 19027.783} C_VEL
LIN {X 0,Y 413.788,Z 860.985,A -85,B 0,C 180,E1 19026.302,E2 19026.302} C_VEL
LIN {X 0,Y 410.568,Z 879.497,A -85,B 0,C 180,E1 19024.573,E2 19024.573} C_VEL
LIN {X 0,Y 407.345,Z 896.813,A -85,B 0,C 180,E1 19022.657,E2 19022.657} C_VEL
LIN {X 0,Y 404.18,Z 913.5,A -85,B 0,C 180,E1 19020.475,E2 19020.475} C_VEL
LIN {X 0,Y 401.25,Z 929.035,A -85,B 0,C 180,E1 19018.099,E2 19018.099} C_VEL
LIN {X 0,Y 398.576,Z 943.871,A -85,B 0,C 180,E1 19015.434,E2 19015.434} C_VEL
LIN {X 0,Y 396.329,Z 957.182,A -85,B 0,C 180,E1 19012.581,E2 19012.581} C_VEL
LIN {X 0,Y 394.645,Z 968.539,A -85,B 0,C 180,E1 19009.695,E2 19009.695} C_VEL
LIN {X 0,Y 393.433,Z 978.436,A -85,B 0,C 180,E1 19006.692,E2 19006.692} C_VEL
LIN {X 0,Y 392.662,Z 986.428,A -85,B 0,C 180,E1 19003.701,E2 19003.701} C_VEL
LIN {X 0,Y 392.234,Z 992.991,A -85,B 0,C 180,E1 19000.579,E2 19000.579} C_VEL
LIN {X 0,Y 392.039,Z 997.687,A -85,B 0,C 180,E1 18997.624,E2 18997.624} C_VEL
LIN {X 0,Y 392.011,Z 1000.723,A -85,B 0,C 180,E1 18994.685,E2 18994.685} C_VEL
LIN {X 0,Y 392.023,Z 1002.377,A -85,B 0,C 180,E1 18991.757,E2 18991.757} C_VEL
LIN {X 0,Y 392.027,Z 1002.486,A -85,B 0,C 180,E1 18988.98,E2 18988.98} C_VEL
LIN {X 0,Y 392.022,Z 1001.264,A -85,B 0,C 180,E1 18986.055,E2 18986.055} C_VEL
LIN {X 0,Y 392.05,Z 998.444,A -85,B 0,C 180,E1 18983.119,E2 18983.119} C_VEL
LIN {X 0,Y 392.173,Z 993.912,A -85,B 0,C 180,E1 18980.02,E2 18980.02} C_VEL
LIN {X 0,Y 392.5,Z 988.279,A -85,B 0,C 180,E1 18977.199,E2 18977.199} C_VEL
LIN {X 0,Y 393.198,Z 980.267,A -85,B 0,C 180,E1 18974.064,E2 18974.064} C_VEL
LIN {X 0,Y 394.278,Z 970.835,A -85,B 0,C 180,E1 18971.063,E2 18971.063} C_VEL
LIN {X 0,Y 395.785,Z 959.964,A -85,B 0,C 180,E1 18968.204,E2 18968.204} C_VEL
LIN {X 0,Y 397.718,Z 947.774,A -85,B 0,C 180,E1 18965.497,E2 18965.497} C_VEL
LIN {X 0,Y 400.051,Z 934.409,A -85,B 0,C 180,E1 18962.947,E2 18962.947} C_VEL
LIN {X 0,Y 402.809,Z 919.22,A -85,B 0,C 180,E1 18960.485,E2 18960.485} C_VEL
LIN {X 0,Y 405.924,Z 902.58,A -85,B 0,C 180,E1 18958.188,E2 18958.188} C_VEL
LIN {X 0,Y 409.263,Z 884.521,A -85,B 0,C 180,E1 18956.071,E2 18956.071} C_VEL
LIN {X 0,Y 412.667,Z 865.539,A -85,B 0,C 180,E1 18954.192,E2 18954.192} C_VEL
LIN {X 0,Y 415.799,Z 846.578,A -85,B 0,C 180,E1 18952.641,E2 18952.641} C_VEL
LIN {X 0,Y 418.929,Z 825.82,A -85,B 0,C 180,E1 18951.239,E2 18951.239} C_VEL
LIN {X 0,Y 421.619,Z 805.623,A -85,B 0,C 180,E1 18950.138,E2 18950.138} C_VEL
LIN {X 0,Y 423.874,Z 784.881,A -85,B 0,C 180,E1 18949.262,E2 18949.262} C_VEL
LIN {X 0,Y 425.756,Z 762.656,A -85,B 0,C 180,E1 18948.578,E2 18948.578} C_VEL
LIN {X 0,Y 426.941,Z 738.056,A -85,B 0,C 180,E1 18948.062,E2 18948.062} C_VEL
LIN {X 0,Y 433.891,Z 522.224,A -85,B 0,C 180,E1 18944.141,E2 18944.141} C_VEL
LIN {X 0,Y 434.763,Z 492.369,A -85,B 0,C 180,E1 18943.565,E2 18943.565} C_VEL
LIN {X 0,Y 434.102,Z 488.537,A -85,B 0,C 180,E1 18943.389,E2 18943.389} C_VEL
LIN {X 0,Y 423.875,Z 471.006,A -85,B 0,C 180,E1 18941.539,E2 18941.539} C_VEL
LIN {X 0,Y 414.018,Z 455.829,A -85,B 0,C 180,E1 18939.61,E2 18939.61} C_VEL
LIN {X 0,Y 412.516,Z 452.97,A -85,B 0,C 180,E1 18939.146,E2 18939.146} C_VEL
LIN {X 0,Y 406.462,Z 440.694,A -85,B 0,C 180,E1 18936.533,E2 18936.533} C_VEL
LIN {X 0,Y 401.172,Z 430.975,A -85,B 0,C 180,E1 18934.109,E2 18934.109} C_VEL
LIN {X 0,Y 398.627,Z 426.359,A -85,B 0,C 180,E1 18932.84,E2 18932.84} C_VEL
LIN {X 0,Y 396.686,Z 422.728,A -85,B 0,C 180,E1 18931.788,E2 18931.788} C_VEL
LIN {X 0,Y 393.924,Z 418.386,A -85,B 0,C 180,E1 18930.338,E2 18930.338} C_VEL
LIN {X 0,Y 393.598,Z 416.918,A -85,B 0,C 180,E1 18929.861,E2 18929.861} C_VEL
LIN {X 0,Y 393.545,Z 416.707,A -85,B 0,C 180,E1 18925.912,E2 18925.912} C_VEL
LIN {X 0,Y 393.531,Z 416.712,A -85,B 0,C 180,E1 18921.93,E2 18921.93} C_VEL
LIN {X 0,Y 393.508,Z 416.707,A -85,B 0,C 180,E1 18918.058,E2 18918.058} C_VEL
LIN {X 0,Y 393.486,Z 416.709,A -85,B 0,C 180,E1 18914.269,E2 18914.269} C_VEL
LIN {X 0,Y 393.49,Z 416.717,A -85,B 0,C 180,E1 18910.393,E2 18910.393} C_VEL
LIN {X 0,Y 393.5,Z 416.72,A -85,B 0,C 180,E1 18906.419,E2 18906.419} C_VEL
LIN {X 0,Y 393.509,Z 416.707,A -85,B 0,C 180,E1 18902.475,E2 18902.475} C_VEL
LIN {X 0,Y 393.532,Z 416.705,A -85,B 0,C 180,E1 18898.689,E2 18898.689} C_VEL
LIN {X 0,Y 393.548,Z 416.715,A -85,B 0,C 180,E1 18894.752,E2 18894.752} C_VEL
LIN {X 0,Y 393.57,Z 416.968,A -85,B 0,C 180,E1 18892.408,E2 18892.408} C_VEL
LIN {X 0,Y 395.013,Z 420.415,A -85,B 0,C 180,E1 18891.264,E2 18891.264} C_VEL
LIN {X 0,Y 396.391,Z 422.281,A -85,B 0,C 180,E1 18890.563,E2 18890.563} C_VEL
LIN {X 0,Y 398.259,Z 425.99,A -85,B 0,C 180,E1 18889.439,E2 18889.439} C_VEL
LIN {X 0,Y 399.246,Z 427.879,A -85,B 0,C 180,E1 18888.881,E2 18888.881} C_VEL
LIN {X 0,Y 401.808,Z 432.78,A -85,B 0,C 180,E1 18887.497,E2 18887.497} C_VEL
LIN {X 0,Y 405.808,Z 440.703,A -85,B 0,C 180,E1 18885.444,E2 18885.444} C_VEL
LIN {X 0,Y 411.605,Z 453.272,A -85,B 0,C 180,E1 18882.598,E2 18882.598} C_VEL
LIN {X 0,Y 421.468,Z 468.534,A -85,B 0,C 180,E1 18880.566,E2 18880.566} C_VEL
LIN {X 0,Y 431.769,Z 485.775,A -85,B 0,C 180,E1 18878.627,E2 18878.627} C_VEL
LIN {X 0,Y 432.678,Z 492.659,A -85,B 0,C 180,E1 18878.329,E2 18878.329} C_VEL
LIN {X 0,Y 423.418,Z 722.594,A -85,B 0,C 180,E1 18873.919,E2 18873.919} C_VEL
LIN {X 0,Y 421.9,Z 743.547,A -85,B 0,C 180,E1 18873.272,E2 18873.272} C_VEL
LIN {X 0,Y 419.9,Z 763.728,A -85,B 0,C 180,E1 18872.402,E2 18872.402} C_VEL
LIN {X 0,Y 417.5,Z 783.375,A -85,B 0,C 180,E1 18871.295,E2 18871.295} C_VEL
LIN {X 0,Y 414.806,Z 801.919,A -85,B 0,C 180,E1 18869.989,E2 18869.989} C_VEL
LIN {X 0,Y 411.847,Z 819.921,A -85,B 0,C 180,E1 18868.436,E2 18868.436} C_VEL
LIN {X 0,Y 408.687,Z 837.452,A -85,B 0,C 180,E1 18866.601,E2 18866.601} C_VEL
LIN {X 0,Y 405.62,Z 853.268,A -85,B 0,C 180,E1 18864.6,E2 18864.6} C_VEL
LIN {X 0,Y 402.799,Z 867.273,A -85,B 0,C 180,E1 18862.494,E2 18862.494} C_VEL
LIN {X 0,Y 400.045,Z 881.022,A -85,B 0,C 180,E1 18860.033,E2 18860.033} C_VEL
LIN {X 0,Y 397.701,Z 893.086,A -85,B 0,C 180,E1 18857.439,E2 18857.439} C_VEL
LIN {X 0,Y 395.838,Z 903.332,A -85,B 0,C 180,E1 18854.782,E2 18854.782} C_VEL
LIN {X 0,Y 394.326,Z 912.594,A -85,B 0,C 180,E1 18851.82,E2 18851.82} C_VEL
LIN {X 0,Y 393.261,Z 920.24,A -85,B 0,C 180,E1 18848.689,E2 18848.689} C_VEL
LIN {X 0,Y 392.673,Z 925.712,A -85,B 0,C 180,E1 18845.664,E2 18845.664} C_VEL
LIN {X 0,Y 392.356,Z 929.424,A -85,B 0,C 180,E1 18842.696,E2 18842.696} C_VEL
LIN {X 0,Y 392.234,Z 931.622,A -85,B 0,C 180,E1 18839.627,E2 18839.627} C_VEL
LIN {X 0,Y 392.202,Z 932.234,A -85,B 0,C 180,E1 18837.068,E2 18837.068} C_VEL
LIN {X 0,Y 391.227,Z 932.272,A -85,B 0,C 180,E1 18835.943,E2 18835.943} C_VEL
LIN {X 0,Y 386.652,Z 931.82,A -85,B 0,C 180,E1 18833.82,E2 18833.82} C_VEL
LIN {X 0,Y 384.472,Z 931.013,A -85,B 0,C 180,E1 18832.361,E2 18832.361} C_VEL
LIN {X 0,Y 384.346,Z 930.709,A -85,B 0,C 180,E1 18831.947,E2 18831.947} C_VEL
LIN {X 0,Y 384.574,Z 927.302,A -85,B 0,C 180,E1 18828.961,E2 18828.961} C_VEL
LIN {X 0,Y 385.067,Z 922.327,A -85,B 0,C 180,E1 18825.972,E2 18825.972} C_VEL
LIN {X 0,Y 385.925,Z 915.775,A -85,B 0,C 180,E1 18823.023,E2 18823.023} C_VEL
LIN {X 0,Y 387.215,Z 907.538,A -85,B 0,C 180,E1 18820.109,E2 18820.109} C_VEL
LIN {X 0,Y 389.032,Z 897.34,A -85,B 0,C 180,E1 18817.218,E2 18817.218} C_VEL
LIN {X 0,Y 391.244,Z 885.807,A -85,B 0,C 180,E1 18814.541,E2 18814.541} C_VEL
LIN {X 0,Y 393.855,Z 872.831,A -85,B 0,C 180,E1 18812.034,E2 18812.034} C_VEL
LIN {X 0,Y 396.851,Z 857.968,A -85,B 0,C 180,E1 18809.636,E2 18809.636} C_VEL
LIN {X 0,Y 400.007,Z 841.99,A -85,B 0,C 180,E1 18807.49,E2 18807.49} C_VEL
LIN {X 0,Y 403.118,Z 825.389,A -85,B 0,C 180,E1 18805.63,E2 18805.63} C_VEL
LIN {X 0,Y 406.193,Z 807.559,A -85,B 0,C 180,E1 18803.97,E2 18803.97} C_VEL
LIN {X 0,Y 409.188,Z 787.897,A -85,B 0,C 180,E1 18802.486,E2 18802.486} C_VEL
LIN {X 0,Y 411.657,Z 768.74,A -85,B 0,C 180,E1 18801.336,E2 18801.336} C_VEL
LIN {X 0,Y 413.771,Z 748.513,A -85,B 0,C 180,E1 18800.39,E2 18800.39} C_VEL
LIN {X 0,Y 415.473,Z 727.097,A -85,B 0,C 180,E1 18799.664,E2 18799.664} C_VEL
LIN {X 0,Y 416.645,Z 702.632,A -85,B 0,C 180,E1 18799.121,E2 18799.121} C_VEL
LIN {X 0,Y 424.343,Z 492.138,A -85,B 0,C 180,E1 18795.168,E2 18795.168} C_VEL
LIN {X 0,Y 423.436,Z 487.504,A -85,B 0,C 180,E1 18794.943,E2 18794.943} C_VEL
LIN {X 0,Y 412.36,Z 468.718,A -85,B 0,C 180,E1 18792.991,E2 18792.991} C_VEL
LIN {X 0,Y 402.105,Z 452.67,A -85,B 0,C 180,E1 18791.062,E2 18791.062} C_VEL
LIN {X 0,Y 395.563,Z 438.343,A -85,B 0,C 180,E1 18788.074,E2 18788.074} C_VEL
LIN {X 0,Y 391.415,Z 429.868,A -85,B 0,C 180,E1 18786.136,E2 18786.136} C_VEL
LIN {X 0,Y 389.385,Z 425.84,A -85,B 0,C 180,E1 18785.165,E2 18785.165} C_VEL
LIN {X 0,Y 387.274,Z 421.669,A -85,B 0,C 180,E1 18784.128,E2 18784.128} C_VEL
LIN {X 0,Y 385.663,Z 417.994,A -85,B 0,C 180,E1 18783.183,E2 18783.183} C_VEL
LIN {X 0,Y 385.627,Z 417.703,A -85,B 0,C 180,E1 18780.824,E2 18780.824} C_VEL
LIN {X 0,Y 385.622,Z 417.701,A -85,B 0,C 180,E1 18776.83,E2 18776.83} C_VEL
LIN {X 0,Y 385.621,Z 417.701,A -85,B 0,C 180,E1 18772.751,E2 18772.751} C_VEL
LIN {X 0,Y 385.623,Z 417.7,A -85,B 0,C 180,E1 18768.758,E2 18768.758} C_VEL
LIN {X 0,Y 385.62,Z 417.698,A -85,B 0,C 180,E1 18764.642,E2 18764.642} C_VEL
LIN {X 0,Y 385.619,Z 417.685,A -85,B 0,C 180,E1 18760.559,E2 18760.559} C_VEL
LIN {X 0,Y 385.614,Z 417.674,A -85,B 0,C 180,E1 18756.503,E2 18756.503} C_VEL
LIN {X 0,Y 385.617,Z 417.684,A -85,B 0,C 180,E1 18752.462,E2 18752.462} C_VEL
LIN {X 0,Y 385.618,Z 417.7,A -85,B 0,C 180,E1 18748.477,E2 18748.477} C_VEL
LIN {X 0,Y 385.615,Z 417.684,A -85,B 0,C 180,E1 18744.348,E2 18744.348} C_VEL
LIN {X 0,Y 385.616,Z 417.671,A -85,B 0,C 180,E1 18740.332,E2 18740.332} C_VEL
LIN {X 0,Y 385.618,Z 417.692,A -85,B 0,C 180,E1 18736.262,E2 18736.262} C_VEL
LIN {X 0,Y 385.62,Z 417.697,A -85,B 0,C 180,E1 18732.276,E2 18732.276} C_VEL
LIN {X 0,Y 385.619,Z 417.674,A -85,B 0,C 180,E1 18728.199,E2 18728.199} C_VEL
LIN {X 0,Y 385.615,Z 417.677,A -85,B 0,C 180,E1 18724.164,E2 18724.164} C_VEL
LIN {X 0,Y 385.621,Z 417.699,A -85,B 0,C 180,E1 18720.149,E2 18720.149} C_VEL
LIN {X 0,Y 385.614,Z 417.693,A -85,B 0,C 180,E1 18716.135,E2 18716.135} C_VEL
LIN {X 0,Y 385.609,Z 417.677,A -85,B 0,C 180,E1 18712.102,E2 18712.102} C_VEL
LIN {X 0,Y 385.611,Z 417.679,A -85,B 0,C 180,E1 18708.028,E2 18708.028} C_VEL
LIN {X 0,Y 385.612,Z 417.684,A -85,B 0,C 180,E1 18704.047,E2 18704.047} C_VEL
LIN {X 0,Y 385.614,Z 417.688,A -85,B 0,C 180,E1 18699.986,E2 18699.986} C_VEL
LIN {X 0,Y 385.615,Z 417.689,A -85,B 0,C 180,E1 18695.979,E2 18695.979} C_VEL
LIN {X 0,Y 385.624,Z 417.685,A -85,B 0,C 180,E1 18692.011,E2 18692.011} C_VEL
LIN {X 0,Y 385.658,Z 418.011,A -85,B 0,C 180,E1 18689.578,E2 18689.578} C_VEL
LIN {X 0,Y 387.122,Z 421.445,A -85,B 0,C 180,E1 18688.726,E2 18688.726} C_VEL
LIN {X 0,Y 388.229,Z 422.878,A -85,B 0,C 180,E1 18688.306,E2 18688.306} C_VEL
LIN {X 0,Y 390.082,Z 426.665,A -85,B 0,C 180,E1 18687.434,E2 18687.434} C_VEL
LIN {X 0,Y 395.798,Z 437.385,A -85,B 0,C 180,E1 18685.01,E2 18685.01} C_VEL
LIN {X 0,Y 402.434,Z 450.569,A -85,B 0,C 180,E1 18682.325,E2 18682.325} C_VEL
LIN {X 0,Y 404.891,Z 455.349,A -85,B 0,C 180,E1 18681.471,E2 18681.471} C_VEL
LIN {X 0,Y 417.137,Z 473.928,A -85,B 0,C 180,E1 18679.197,E2 18679.197} C_VEL
LIN {X 0,Y 428.906,Z 493.508,A -85,B 0,C 180,E1 18677.159,E2 18677.159} C_VEL
LIN {X 0,Y 428.811,Z 502.286,A -85,B 0,C 180,E1 18676.968,E2 18676.968} C_VEL
LIN {X 0,Y 421.392,Z 722.942,A -85,B 0,C 180,E1 18672.928,E2 18672.928} C_VEL
LIN {X 0,Y 419.999,Z 759.011,A -85,B 0,C 180,E1 18672.231,E2 18672.231} C_VEL
LIN {X 0,Y 418.192,Z 780.881,A -85,B 0,C 180,E1 18671.603,E2 18671.603} C_VEL
LIN {X 0,Y 415.889,Z 801.963,A -85,B 0,C 180,E1 18670.75,E2 18670.75} C_VEL
LIN {X 0,Y 413.084,Z 823.284,A -85,B 0,C 180,E1 18669.63,E2 18669.63} C_VEL
LIN {X 0,Y 410.054,Z 843.069,A -85,B 0,C 180,E1 18668.335,E2 18668.335} C_VEL
LIN {X 0,Y 406.673,Z 862.389,A -85,B 0,C 180,E1 18666.778,E2 18666.778} C_VEL
LIN {X 0,Y 403.051,Z 881.931,A -85,B 0,C 180,E1 18664.879,E2 18664.879} C_VEL
LIN {X 0,Y 399.65,Z 899.268,A -85,B 0,C 180,E1 18662.884,E2 18662.884} C_VEL
LIN {X 0,Y 396.369,Z 915.738,A -85,B 0,C 180,E1 18660.637,E2 18660.637} C_VEL
LIN {X 0,Y 393.356,Z 930.827,A -85,B 0,C 180,E1 18658.218,E2 18658.218} C_VEL
LIN {X 0,Y 390.726,Z 944.68,A -85,B 0,C 180,E1 18655.627,E2 18655.627} C_VEL
LIN {X 0,Y 388.513,Z 957.18,A -85,B 0,C 180,E1 18652.87,E2 18652.87} C_VEL
LIN {X 0,Y 386.761,Z 968.314,A -85,B 0,C 180,E1 18649.956,E2 18649.956} C_VEL
LIN {X 0,Y 385.472,Z 978.264,A -85,B 0,C 180,E1 18646.839,E2 18646.839} C_VEL
LIN {X 0,Y 384.686,Z 986.066,A -85,B 0,C 180,E1 18643.838,E2 18643.838} C_VEL
LIN {X 0,Y 384.263,Z 992.269,A -85,B 0,C 180,E1 18640.801,E2 18640.801} C_VEL
LIN {X 0,Y 384.064,Z 996.973,A -85,B 0,C 180,E1 18637.783,E2 18637.783} C_VEL
LIN {X 0,Y 384.034,Z 1000.01,A -85,B 0,C 180,E1 18634.782,E2 18634.782} C_VEL
LIN {X 0,Y 384.053,Z 1001.667,A -85,B 0,C 180,E1 18631.793,E2 18631.793} C_VEL
LIN {X 0,Y 384.059,Z 1001.769,A -85,B 0,C 180,E1 18628.959,E2 18628.959} C_VEL
LIN {X 0,Y 384.049,Z 1000.539,A -85,B 0,C 180,E1 18625.972,E2 18625.972} C_VEL
LIN {X 0,Y 384.067,Z 997.705,A -85,B 0,C 180,E1 18622.975,E2 18622.975} C_VEL
LIN {X 0,Y 384.203,Z 993.156,A -85,B 0,C 180,E1 18619.811,E2 18619.811} C_VEL
LIN {X 0,Y 384.547,Z 987.506,A -85,B 0,C 180,E1 18616.93,E2 18616.93} C_VEL
LIN {X 0,Y 385.288,Z 979.474,A -85,B 0,C 180,E1 18613.727,E2 18613.727} C_VEL
LIN {X 0,Y 386.446,Z 970.016,A -85,B 0,C 180,E1 18610.664,E2 18610.664} C_VEL
LIN {X 0,Y 388.056,Z 959.125,A -85,B 0,C 180,E1 18607.747,E2 18607.747} C_VEL
LIN {X 0,Y 390.116,Z 946.908,A -85,B 0,C 180,E1 18604.987,E2 18604.987} C_VEL
LIN {X 0,Y 392.605,Z 933.524,A -85,B 0,C 180,E1 18602.391,E2 18602.391} C_VEL
LIN {X 0,Y 395.54,Z 918.312,A -85,B 0,C 180,E1 18599.887,E2 18599.887} C_VEL
LIN {X 0,Y 398.818,Z 901.673,A -85,B 0,C 180,E1 18597.558,E2 18597.558} C_VEL
LIN {X 0,Y 402.371,Z 883.552,A -85,B 0,C 180,E1 18595.408,E2 18595.408} C_VEL
LIN {X 0,Y 405.803,Z 865.307,A -85,B 0,C 180,E1 18593.578,E2 18593.578} C_VEL
LIN {X 0,Y 409.126,Z 846.19,A -85,B 0,C 180,E1 18591.991,E2 18591.991} C_VEL
LIN {X 0,Y 412.422,Z 825.463,A -85,B 0,C 180,E1 18590.572,E2 18590.572} C_VEL
LIN {X 0,Y 415.246,Z 805.237,A -85,B 0,C 180,E1 18589.454,E2 18589.454} C_VEL
LIN {X 0,Y 417.635,Z 784.181,A -85,B 0,C 180,E1 18588.559,E2 18588.559} C_VEL
LIN {X 0,Y 419.59,Z 762.103,A -85,B 0,C 180,E1 18587.877,E2 18587.877} C_VEL
LIN {X 0,Y 420.823,Z 737.332,A -85,B 0,C 180,E1 18587.353,E2 18587.353} C_VEL
LIN {X 0,Y 428.262,Z 519.925,A -85,B 0,C 180,E1 18583.349,E2 18583.349} C_VEL
LIN {X 0,Y 429.065,Z 493.761,A -85,B 0,C 180,E1 18582.833,E2 18582.833} C_VEL
LIN {X 0,Y 428.374,Z 491.808,A -85,B 0,C 180,E1 18582.691,E2 18582.691} C_VEL
LIN {X 0,Y 418.548,Z 475.017,A -85,B 0,C 180,E1 18580.84,E2 18580.84} C_VEL
LIN {X 0,Y 409.031,Z 460.232,A -85,B 0,C 180,E1 18578.896,E2 18578.896} C_VEL
LIN {X 0,Y 404.914,Z 454.022,A -85,B 0,C 180,E1 18577.941,E2 18577.941} C_VEL
LIN {X 0,Y 398.953,Z 442.019,A -85,B 0,C 180,E1 18575.199,E2 18575.199} C_VEL
LIN {X 0,Y 393.962,Z 432.808,A -85,B 0,C 180,E1 18572.723,E2 18572.723} C_VEL
LIN {X 0,Y 391.766,Z 428.83,A -85,B 0,C 180,E1 18571.532,E2 18571.532} C_VEL
LIN {X 0,Y 389.004,Z 424.232,A -85,B 0,C 180,E1 18569.99,E2 18569.99} C_VEL
LIN {X 0,Y 388.187,Z 422.691,A -85,B 0,C 180,E1 18569.469,E2 18569.469} C_VEL
LIN {X 0,Y 386.128,Z 419.756,A -85,B 0,C 180,E1 18568.285,E2 18568.285} C_VEL
LIN {X 0,Y 385.635,Z 417.901,A -85,B 0,C 180,E1 18567.597,E2 18567.597} C_VEL
LIN {X 0,Y 385.61,Z 417.691,A -85,B 0,C 180,E1 18563.697,E2 18563.697} C_VEL
LIN {X 0,Y 385.599,Z 417.701,A -85,B 0,C 180,E1 18559.699,E2 18559.699} C_VEL
LIN {X 0,Y 385.593,Z 417.698,A -85,B 0,C 180,E1 18555.645,E2 18555.645} C_VEL
LIN {X 0,Y 385.58,Z 417.693,A -85,B 0,C 180,E1 18551.669,E2 18551.669} C_VEL
LIN {X 0,Y 385.58,Z 417.694,A -85,B 0,C 180,E1 18547.749,E2 18547.749} C_VEL
LIN {X 0,Y 385.572,Z 417.706,A -85,B 0,C 180,E1 18543.866,E2 18543.866} C_VEL
LIN {X 0,Y 385.573,Z 417.701,A -85,B 0,C 180,E1 18540,E2 18540} C_VEL
LIN {X 0,Y 385.577,Z 417.696,A -85,B 0,C 180,E1 18535.985,E2 18535.985} C_VEL
LIN {X 0,Y 385.66,Z 418.109,A -85,B 0,C 180,E1 18534.57,E2 18534.57} C_VEL
LIN {X 0,Y 387.122,Z 421.472,A -85,B 0,C 180,E1 18533.325,E2 18533.325} C_VEL
LIN {X 0,Y 388.613,Z 423.501,A -85,B 0,C 180,E1 18532.46,E2 18532.46} C_VEL
LIN {X 0,Y 390.608,Z 427.266,A -85,B 0,C 180,E1 18531.165,E2 18531.165} C_VEL
LIN {X 0,Y 391.734,Z 429.539,A -85,B 0,C 180,E1 18530.45,E2 18530.45} C_VEL
LIN {X 0,Y 393.973,Z 433.541,A -85,B 0,C 180,E1 18529.175,E2 18529.175} C_VEL
LIN {X 0,Y 398.296,Z 441.973,A -85,B 0,C 180,E1 18526.794,E2 18526.794} C_VEL
LIN {X 0,Y 403.637,Z 453.264,A -85,B 0,C 180,E1 18524.04,E2 18524.04} C_VEL
LIN {X 0,Y 413.935,Z 468.883,A -85,B 0,C 180,E1 18521.753,E2 18521.753} C_VEL
LIN {X 0,Y 423.937,Z 485.412,A -85,B 0,C 180,E1 18519.75,E2 18519.75} C_VEL
LIN {X 0,Y 426.737,Z 490.678,A -85,B 0,C 180,E1 18519.208,E2 18519.208} C_VEL
LIN {X 0,Y 427.036,Z 494.677,A -85,B 0,C 180,E1 18519.062,E2 18519.062} C_VEL
LIN {X 0,Y 417.327,Z 723.048,A -85,B 0,C 180,E1 18514.623,E2 18514.623} C_VEL
LIN {X 0,Y 415.749,Z 743.879,A -85,B 0,C 180,E1 18513.973,E2 18513.973} C_VEL
LIN {X 0,Y 413.669,Z 763.932,A -85,B 0,C 180,E1 18513.102,E2 18513.102} C_VEL
LIN {X 0,Y 411.134,Z 783.809,A -85,B 0,C 180,E1 18511.972,E2 18511.972} C_VEL
LIN {X 0,Y 408.318,Z 802.368,A -85,B 0,C 180,E1 18510.653,E2 18510.653} C_VEL
LIN {X 0,Y 405.294,Z 819.954,A -85,B 0,C 180,E1 18509.127,E2 18509.127} C_VEL
LIN {X 0,Y 402.081,Z 836.858,A -85,B 0,C 180,E1 18507.342,E2 18507.342} C_VEL
LIN {X 0,Y 398.804,Z 852.908,A -85,B 0,C 180,E1 18505.311,E2 18505.311} C_VEL
LIN {X 0,Y 395.697,Z 867.615,A -85,B 0,C 180,E1 18503.086,E2 18503.086} C_VEL
LIN {X 0,Y 392.796,Z 881.267,A -85,B 0,C 180,E1 18500.615,E2 18500.615} C_VEL
LIN {X 0,Y 390.338,Z 893.125,A -85,B 0,C 180,E1 18498.044,E2 18498.044} C_VEL
LIN {X 0,Y 388.272,Z 903.661,A -85,B 0,C 180,E1 18495.289,E2 18495.289} C_VEL
LIN {X 0,Y 386.607,Z 913.039,A -85,B 0,C 180,E1 18492.248,E2 18492.248} C_VEL
LIN {X 0,Y 385.486,Z 920.285,A -85,B 0,C 180,E1 18489.257,E2 18489.257} C_VEL
LIN {X 0,Y 384.827,Z 925.702,A -85,B 0,C 180,E1 18486.321,E2 18486.321} C_VEL
LIN {X 0,Y 384.44,Z 929.851,A -85,B 0,C 180,E1 18483.126,E2 18483.126} C_VEL
LIN {X 0,Y 384.282,Z 932.163,A -85,B 0,C 180,E1 18480.139,E2 18480.139} C_VEL
LIN {X 0,Y 384.235,Z 932.952,A -85,B 0,C 180,E1 18477.085,E2 18477.085} C_VEL
LIN {X 0,Y 384.258,Z 932.158,A -85,B 0,C 180,E1 18474.108,E2 18474.108} C_VEL
LIN {X 0,Y 384.346,Z 930.709,A -85,B 0,C 180,E1 18471.947,E2 18471.947} C_VEL
LIN {X 0,Y 383.417,Z 929.78,A -85,B 0,C 180,E1 18470.805,E2 18470.805} C_VEL
LIN {X 0,Y 377.433,Z 926.32,A -85,B 0,C 180,E1 18467.683,E2 18467.683} C_VEL
LIN {X 0,Y 376.962,Z 924.919,A -85,B 0,C 180,E1 18466.777,E2 18466.777} C_VEL
LIN {X 0,Y 377.743,Z 918.818,A -85,B 0,C 180,E1 18463.729,E2 18463.729} C_VEL
LIN {X 0,Y 379.019,Z 910.806,A -85,B 0,C 180,E1 18460.638,E2 18460.638} C_VEL
LIN {X 0,Y 380.779,Z 901.242,A -85,B 0,C 180,E1 18457.693,E2 18457.693} C_VEL
LIN {X 0,Y 382.983,Z 890.332,A -85,B 0,C 180,E1 18454.939,E2 18454.939} C_VEL
LIN {X 0,Y 385.58,Z 878.105,A -85,B 0,C 180,E1 18452.375,E2 18452.375} C_VEL
LIN {X 0,Y 388.478,Z 864.474,A -85,B 0,C 180,E1 18449.997,E2 18449.997} C_VEL
LIN {X 0,Y 391.614,Z 849.499,A -85,B 0,C 180,E1 18447.802,E2 18447.802} C_VEL
LIN {X 0,Y 394.92,Z 833.053,A -85,B 0,C 180,E1 18445.786,E2 18445.786} C_VEL
LIN {X 0,Y 398.162,Z 815.683,A -85,B 0,C 180,E1 18444.015,E2 18444.015} C_VEL
LIN {X 0,Y 401.273,Z 797.407,A -85,B 0,C 180,E1 18442.48,E2 18442.48} C_VEL
LIN {X 0,Y 404.088,Z 778.145,A -85,B 0,C 180,E1 18441.173,E2 18441.173} C_VEL
LIN {X 0,Y 406.492,Z 758.328,A -85,B 0,C 180,E1 18440.118,E2 18440.118} C_VEL
LIN {X 0,Y 408.446,Z 737.91,A -85,B 0,C 180,E1 18439.298,E2 18439.298} C_VEL
LIN {X 0,Y 409.892,Z 715.898,A -85,B 0,C 180,E1 18438.683,E2 18438.683} C_VEL
LIN {X 0,Y 418.498,Z 493.76,A -85,B 0,C 180,E1 18434.448,E2 18434.448} C_VEL
LIN {X 0,Y 417.873,Z 491.343,A -85,B 0,C 180,E1 18434.306,E2 18434.306} C_VEL
LIN {X 0,Y 407.308,Z 473.439,A -85,B 0,C 180,E1 18432.394,E2 18432.394} C_VEL
LIN {X 0,Y 396.388,Z 456.402,A -85,B 0,C 180,E1 18430.281,E2 18430.281} C_VEL
LIN {X 0,Y 393.891,Z 452.404,A -85,B 0,C 180,E1 18429.724,E2 18429.724} C_VEL
LIN {X 0,Y 387.498,Z 438.844,A -85,B 0,C 180,E1 18426.721,E2 18426.721} C_VEL
LIN {X 0,Y 383.678,Z 431.132,A -85,B 0,C 180,E1 18424.861,E2 18424.861} C_VEL
LIN {X 0,Y 381.75,Z 427.28,A -85,B 0,C 180,E1 18423.892,E2 18423.892} C_VEL
LIN {X 0,Y 379.321,Z 422.614,A -85,B 0,C 180,E1 18422.662,E2 18422.662} C_VEL
LIN {X 0,Y 377.702,Z 418.887,A -85,B 0,C 180,E1 18421.617,E2 18421.617} C_VEL
LIN {X 0,Y 377.674,Z 418.683,A -85,B 0,C 180,E1 18417.669,E2 18417.669} C_VEL
LIN {X 0,Y 377.676,Z 418.685,A -85,B 0,C 180,E1 18413.593,E2 18413.593} C_VEL
LIN {X 0,Y 377.68,Z 418.679,A -85,B 0,C 180,E1 18409.561,E2 18409.561} C_VEL
LIN {X 0,Y 377.676,Z 418.672,A -85,B 0,C 180,E1 18405.411,E2 18405.411} C_VEL
LIN {X 0,Y 377.685,Z 418.663,A -85,B 0,C 180,E1 18401.44,E2 18401.44} C_VEL
LIN {X 0,Y 377.68,Z 418.666,A -85,B 0,C 180,E1 18397.416,E2 18397.416} C_VEL
LIN {X 0,Y 377.682,Z 418.687,A -85,B 0,C 180,E1 18393.412,E2 18393.412} C_VEL
LIN {X 0,Y 377.683,Z 418.683,A -85,B 0,C 180,E1 18389.325,E2 18389.325} C_VEL
LIN {X 0,Y 377.677,Z 418.659,A -85,B 0,C 180,E1 18385.229,E2 18385.229} C_VEL
LIN {X 0,Y 377.678,Z 418.668,A -85,B 0,C 180,E1 18381.266,E2 18381.266} C_VEL
LIN {X 0,Y 377.679,Z 418.69,A -85,B 0,C 180,E1 18377.09,E2 18377.09} C_VEL
LIN {X 0,Y 377.676,Z 418.676,A -85,B 0,C 180,E1 18373.005,E2 18373.005} C_VEL
LIN {X 0,Y 377.675,Z 418.661,A -85,B 0,C 180,E1 18368.987,E2 18368.987} C_VEL
LIN {X 0,Y 377.68,Z 418.681,A -85,B 0,C 180,E1 18365.012,E2 18365.012} C_VEL
LIN {X 0,Y 377.684,Z 418.686,A -85,B 0,C 180,E1 18360.911,E2 18360.911} C_VEL
LIN {X 0,Y 377.677,Z 418.67,A -85,B 0,C 180,E1 18356.813,E2 18356.813} C_VEL
LIN {X 0,Y 377.686,Z 418.661,A -85,B 0,C 180,E1 18352.7,E2 18352.7} C_VEL
LIN {X 0,Y 377.679,Z 418.669,A -85,B 0,C 180,E1 18348.548,E2 18348.548} C_VEL
LIN {X 0,Y 377.685,Z 418.677,A -85,B 0,C 180,E1 18344.492,E2 18344.492} C_VEL
LIN {X 0,Y 377.683,Z 418.681,A -85,B 0,C 180,E1 18340.354,E2 18340.354} C_VEL
LIN {X 0,Y 377.685,Z 418.68,A -85,B 0,C 180,E1 18336.272,E2 18336.272} C_VEL
LIN {X 0,Y 377.69,Z 418.674,A -85,B 0,C 180,E1 18332.156,E2 18332.156} C_VEL
LIN {X 0,Y 377.751,Z 419.127,A -85,B 0,C 180,E1 18331.083,E2 18331.083} C_VEL
LIN {X 0,Y 379.463,Z 422.795,A -85,B 0,C 180,E1 18330.133,E2 18330.133} C_VEL
LIN {X 0,Y 380.73,Z 425.039,A -85,B 0,C 180,E1 18329.546,E2 18329.546} C_VEL
LIN {X 0,Y 383.292,Z 429.618,A -85,B 0,C 180,E1 18328.377,E2 18328.377} C_VEL
LIN {X 0,Y 388.524,Z 439.521,A -85,B 0,C 180,E1 18326.052,E2 18326.052} C_VEL
LIN {X 0,Y 394.688,Z 451.589,A -85,B 0,C 180,E1 18323.465,E2 18323.465} C_VEL
LIN {X 0,Y 396.797,Z 455.497,A -85,B 0,C 180,E1 18322.744,E2 18322.744} C_VEL
LIN {X 0,Y 409.587,Z 474.688,A -85,B 0,C 180,E1 18320.261,E2 18320.261} C_VEL
LIN {X 0,Y 421.523,Z 494.135,A -85,B 0,C 180,E1 18318.109,E2 18318.109} C_VEL
LIN {X 0,Y 423.208,Z 497.437,A -85,B 0,C 180,E1 18317.806,E2 18317.806} C_VEL
LIN {X 0,Y 415.561,Z 713.38,A -85,B 0,C 180,E1 18313.808,E2 18313.808} C_VEL
LIN {X 0,Y 413.874,Z 757.723,A -85,B 0,C 180,E1 18312.957,E2 18312.957} C_VEL
LIN {X 0,Y 412.005,Z 779.629,A -85,B 0,C 180,E1 18312.329,E2 18312.329} C_VEL
LIN {X 0,Y 409.66,Z 800.405,A -85,B 0,C 180,E1 18311.495,E2 18311.495} C_VEL
LIN {X 0,Y 406.934,Z 820.701,A -85,B 0,C 180,E1 18310.443,E2 18310.443} C_VEL
LIN {X 0,Y 403.798,Z 840.426,A -85,B 0,C 180,E1 18309.157,E2 18309.157} C_VEL
LIN {X 0,Y 400.193,Z 860.389,A -85,B 0,C 180,E1 18307.564,E2 18307.564} C_VEL
LIN {X 0,Y 396.491,Z 879.62,A -85,B 0,C 180,E1 18305.708,E2 18305.708} C_VEL
LIN {X 0,Y 392.89,Z 897.301,A -85,B 0,C 180,E1 18303.678,E2 18303.678} C_VEL
LIN {X 0,Y 389.282,Z 914.297,A -85,B 0,C 180,E1 18301.343,E2 18301.343} C_VEL
LIN {X 0,Y 385.991,Z 929.959,A -85,B 0,C 180,E1 18298.806,E2 18298.806} C_VEL
LIN {X 0,Y 383.192,Z 943.913,A -85,B 0,C 180,E1 18296.157,E2 18296.157} C_VEL
LIN {X 0,Y 380.841,Z 956.391,A -85,B 0,C 180,E1 18293.358,E2 18293.358} C_VEL
LIN {X 0,Y 378.968,Z 967.547,A -85,B 0,C 180,E1 18290.384,E2 18290.384} C_VEL
LIN {X 0,Y 377.599,Z 977.371,A -85,B 0,C 180,E1 18287.254,E2 18287.254} C_VEL
LIN {X 0,Y 376.77,Z 984.957,A -85,B 0,C 180,E1 18284.291,E2 18284.291} C_VEL
LIN {X 0,Y 376.289,Z 991.546,A -85,B 0,C 180,E1 18281.033,E2 18281.033} C_VEL
LIN {X 0,Y 376.092,Z 996.26,A -85,B 0,C 180,E1 18277.949,E2 18277.949} C_VEL
LIN {X 0,Y 376.057,Z 999.298,A -85,B 0,C 180,E1 18274.884,E2 18274.884} C_VEL
LIN {X 0,Y 376.084,Z 1000.956,A -85,B 0,C 180,E1 18271.831,E2 18271.831} C_VEL
LIN {X 0,Y 376.091,Z 1001.052,A -85,B 0,C 180,E1 18268.937,E2 18268.937} C_VEL
LIN {X 0,Y 376.076,Z 999.814,A -85,B 0,C 180,E1 18265.887,E2 18265.887} C_VEL
LIN {X 0,Y 376.086,Z 997.139,A -85,B 0,C 180,E1 18262.979,E2 18262.979} C_VEL
LIN {X 0,Y 376.202,Z 992.943,A -85,B 0,C 180,E1 18259.901,E2 18259.901} C_VEL
LIN {X 0,Y 376.571,Z 987.065,A -85,B 0,C 180,E1 18256.804,E2 18256.804} C_VEL
LIN {X 0,Y 377.338,Z 979.113,A -85,B 0,C 180,E1 18253.533,E2 18253.533} C_VEL
LIN {X 0,Y 378.551,Z 969.741,A -85,B 0,C 180,E1 18250.405,E2 18250.405} C_VEL
LIN {X 0,Y 380.3,Z 958.568,A -85,B 0,C 180,E1 18247.341,E2 18247.341} C_VEL
LIN {X 0,Y 382.544,Z 946.059,A -85,B 0,C 180,E1 18244.457,E2 18244.457} C_VEL
LIN {X 0,Y 385.196,Z 932.64,A -85,B 0,C 180,E1 18241.813,E2 18241.813} C_VEL
LIN {X 0,Y 388.428,Z 916.941,A -85,B 0,C 180,E1 18239.191,E2 18239.191} C_VEL
LIN {X 0,Y 391.774,Z 900.755,A -85,B 0,C 180,E1 18236.901,E2 18236.901} C_VEL
LIN {X 0,Y 395.496,Z 882.777,A -85,B 0,C 180,E1 18234.743,E2 18234.743} C_VEL
LIN {X 0,Y 399.143,Z 864.318,A -85,B 0,C 180,E1 18232.869,E2 18232.869} C_VEL
LIN {X 0,Y 402.778,Z 844.463,A -85,B 0,C 180,E1 18231.212,E2 18231.212} C_VEL
LIN {X 0,Y 406.098,Z 824.333,A -85,B 0,C 180,E1 18229.834,E2 18229.834} C_VEL
LIN {X 0,Y 409.04,Z 803.933,A -85,B 0,C 180,E1 18228.707,E2 18228.707} C_VEL
LIN {X 0,Y 411.556,Z 782.738,A -85,B 0,C 180,E1 18227.804,E2 18227.804} C_VEL
LIN {X 0,Y 413.547,Z 761.034,A -85,B 0,C 180,E1 18227.139,E2 18227.139} C_VEL
LIN {X 0,Y 414.872,Z 734.335,A -85,B 0,C 180,E1 18226.576,E2 18226.576} C_VEL
LIN {X 0,Y 422.598,Z 521.338,A -85,B 0,C 180,E1 18222.604,E2 18222.604} C_VEL
LIN {X 0,Y 423.445,Z 496.523,A -85,B 0,C 180,E1 18222.112,E2 18222.112} C_VEL
LIN {X 0,Y 413.744,Z 479.71,A -85,B 0,C 180,E1 18220.209,E2 18220.209} C_VEL
LIN {X 0,Y 404.28,Z 464.908,A -85,B 0,C 180,E1 18218.191,E2 18218.191} C_VEL
LIN {X 0,Y 396.957,Z 454.321,A -85,B 0,C 180,E1 18216.472,E2 18216.472} C_VEL
LIN {X 0,Y 391.59,Z 443.64,A -85,B 0,C 180,E1 18213.822,E2 18213.822} C_VEL
LIN {X 0,Y 388.728,Z 438.535,A -85,B 0,C 180,E1 18212.344,E2 18212.344} C_VEL
LIN {X 0,Y 386.367,Z 434.112,A -85,B 0,C 180,E1 18210.996,E2 18210.996} C_VEL
LIN {X 0,Y 384.107,Z 430.105,A -85,B 0,C 180,E1 18209.642,E2 18209.642} C_VEL
LIN {X 0,Y 381.239,Z 425.404,A -85,B 0,C 180,E1 18207.828,E2 18207.828} C_VEL
LIN {X 0,Y 380.688,Z 424.106,A -85,B 0,C 180,E1 18207.363,E2 18207.363} C_VEL
LIN {X 0,Y 378.364,Z 421.091,A -85,B 0,C 180,E1 18205.85,E2 18205.85} C_VEL
LIN {X 0,Y 377.651,Z 418.864,A -85,B 0,C 180,E1 18204.811,E2 18204.811} C_VEL
LIN {X 0,Y 377.625,Z 418.684,A -85,B 0,C 180,E1 18200.943,E2 18200.943} C_VEL
LIN {X 0,Y 377.62,Z 418.69,A -85,B 0,C 180,E1 18196.933,E2 18196.933} C_VEL
LIN {X 0,Y 377.629,Z 418.698,A -85,B 0,C 180,E1 18193.006,E2 18193.006} C_VEL
LIN {X 0,Y 377.64,Z 418.684,A -85,B 0,C 180,E1 18188.987,E2 18188.987} C_VEL
LIN {X 0,Y 377.663,Z 418.679,A -85,B 0,C 180,E1 18185.164,E2 18185.164} C_VEL
LIN {X 0,Y 377.675,Z 418.685,A -85,B 0,C 180,E1 18181.061,E2 18181.061} C_VEL
LIN {X 0,Y 377.706,Z 418.969,A -85,B 0,C 180,E1 18177.344,E2 18177.344} C_VEL
LIN {X 0,Y 379.416,Z 422.785,A -85,B 0,C 180,E1 18175.617,E2 18175.617} C_VEL
LIN {X 0,Y 380.791,Z 424.469,A -85,B 0,C 180,E1 18174.727,E2 18174.727} C_VEL
LIN {X 0,Y 382.495,Z 427.993,A -85,B 0,C 180,E1 18173.395,E2 18173.395} C_VEL
LIN {X 0,Y 383.7,Z 429.715,A -85,B 0,C 180,E1 18172.664,E2 18172.664} C_VEL
LIN {X 0,Y 385.67,Z 433.454,A -85,B 0,C 180,E1 18171.351,E2 18171.351} C_VEL
LIN {X 0,Y 388.92,Z 439.749,A -85,B 0,C 180,E1 18169.332,E2 18169.332} C_VEL
LIN {X 0,Y 392.934,Z 447.628,A -85,B 0,C 180,E1 18167.06,E2 18167.06} C_VEL
LIN {X 0,Y 395.86,Z 453.869,A -85,B 0,C 180,E1 18165.519,E2 18165.519} C_VEL
LIN {X 0,Y 404.54,Z 466.408,A -85,B 0,C 180,E1 18163.446,E2 18163.446} C_VEL
LIN {X 0,Y 414.552,Z 482.36,A -85,B 0,C 180,E1 18161.271,E2 18161.271} C_VEL
LIN {X 0,Y 421.552,Z 494.829,A -85,B 0,C 180,E1 18159.852,E2 18159.852} C_VEL
LIN {X 0,Y 411.301,Z 723.611,A -85,B 0,C 180,E1 18155.347,E2 18155.347} C_VEL
LIN {X 0,Y 409.645,Z 744.547,A -85,B 0,C 180,E1 18154.685,E2 18154.685} C_VEL
LIN {X 0,Y 407.527,Z 764.12,A -85,B 0,C 180,E1 18153.827,E2 18153.827} C_VEL
LIN {X 0,Y 404.952,Z 783.527,A -85,B 0,C 180,E1 18152.721,E2 18152.721} C_VEL
LIN {X 0,Y 402.005,Z 802.212,A -85,B 0,C 180,E1 18151.389,E2 18151.389} C_VEL
LIN {X 0,Y 398.843,Z 819.746,A -85,B 0,C 180,E1 18149.86,E2 18149.86} C_VEL
LIN {X 0,Y 395.409,Z 837.006,A -85,B 0,C 180,E1 18148.027,E2 18148.027} C_VEL
LIN {X 0,Y 391.981,Z 852.985,A -85,B 0,C 180,E1 18145.988,E2 18145.988} C_VEL
LIN {X 0,Y 388.681,Z 867.808,A -85,B 0,C 180,E1 18143.724,E2 18143.724} C_VEL
LIN {X 0,Y 385.669,Z 881.193,A -85,B 0,C 180,E1 18141.286,E2 18141.286} C_VEL
LIN {X 0,Y 383.007,Z 893.219,A -85,B 0,C 180,E1 18138.664,E2 18138.664} C_VEL
LIN {X 0,Y 380.721,Z 904.035,A -85,B 0,C 180,E1 18135.798,E2 18135.798} C_VEL
LIN {X 0,Y 378.96,Z 913.118,A -85,B 0,C 180,E1 18132.82,E2 18132.82} C_VEL
LIN {X 0,Y 377.739,Z 920.38,A -85,B 0,C 180,E1 18129.828,E2 18129.828} C_VEL
LIN {X 0,Y 376.939,Z 926.278,A -85,B 0,C 180,E1 18126.638,E2 18126.638} C_VEL
LIN {X 0,Y 376.523,Z 930.351,A -85,B 0,C 180,E1 18123.505,E2 18123.505} C_VEL
LIN {X 0,Y 376.332,Z 932.771,A -85,B 0,C 180,E1 18120.49,E2 18120.49} C_VEL
LIN {X 0,Y 376.266,Z 933.63,A -85,B 0,C 180,E1 18117.433,E2 18117.433} C_VEL
LIN {X 0,Y 376.289,Z 932.979,A -85,B 0,C 180,E1 18114.299,E2 18114.299} C_VEL
LIN {X 0,Y 376.413,Z 930.776,A -85,B 0,C 180,E1 18111.173,E2 18111.173} C_VEL
LIN {X 0,Y 376.752,Z 927.034,A -85,B 0,C 180,E1 18108.086,E2 18108.086} C_VEL
LIN {X 0,Y 376.962,Z 924.919,A -85,B 0,C 180,E1 18106.777,E2 18106.777} C_VEL
LIN {X 0,Y 376.229,Z 923.053,A -85,B 0,C 180,E1 18105.636,E2 18105.636} C_VEL
LIN {X 0,Y 370.977,Z 917.431,A -85,B 0,C 180,E1 18102.595,E2 18102.595} C_VEL
LIN {X 0,Y 370.638,Z 915.123,A -85,B 0,C 180,E1 18101.626,E2 18101.626} C_VEL
LIN {X 0,Y 372.234,Z 906.498,A -85,B 0,C 180,E1 18098.648,E2 18098.648} C_VEL
LIN {X 0,Y 374.436,Z 895.852,A -85,B 0,C 180,E1 18095.667,E2 18095.667} C_VEL
LIN {X 0,Y 376.94,Z 884.498,A -85,B 0,C 180,E1 18093.038,E2 18093.038} C_VEL
LIN {X 0,Y 379.973,Z 871.073,A -85,B 0,C 180,E1 18090.449,E2 18090.449} C_VEL
LIN {X 0,Y 383.432,Z 855.594,A -85,B 0,C 180,E1 18087.979,E2 18087.979} C_VEL
LIN {X 0,Y 386.888,Z 839.466,A -85,B 0,C 180,E1 18085.847,E2 18085.847} C_VEL
LIN {X 0,Y 390.301,Z 822.388,A -85,B 0,C 180,E1 18083.968,E2 18083.968} C_VEL
LIN {X 0,Y 393.602,Z 804.398,A -85,B 0,C 180,E1 18082.333,E2 18082.333} C_VEL
LIN {X 0,Y 396.659,Z 785.507,A -85,B 0,C 180,E1 18080.933,E2 18080.933} C_VEL
LIN {X 0,Y 399.242,Z 766.721,A -85,B 0,C 180,E1 18079.812,E2 18079.812} C_VEL
LIN {X 0,Y 401.565,Z 745.57,A -85,B 0,C 180,E1 18078.851,E2 18078.851} C_VEL
LIN {X 0,Y 403.213,Z 725.028,A -85,B 0,C 180,E1 18078.183,E2 18078.183} C_VEL
LIN {X 0,Y 404.614,Z 694.91,A -85,B 0,C 180,E1 18077.544,E2 18077.544} C_VEL
LIN {X 0,Y 412.641,Z 495.694,A -85,B 0,C 180,E1 18073.708,E2 18073.708} C_VEL
LIN {X 0,Y 401.44,Z 476.675,A -85,B 0,C 180,E1 18071.614,E2 18071.614} C_VEL
LIN {X 0,Y 389.371,Z 457.989,A -85,B 0,C 180,E1 18069.182,E2 18069.182} C_VEL
LIN {X 0,Y 385.578,Z 452.301,A -85,B 0,C 180,E1 18068.311,E2 18068.311} C_VEL
LIN {X 0,Y 380.463,Z 441.282,A -85,B 0,C 180,E1 18065.773,E2 18065.773} C_VEL
LIN {X 0,Y 376.157,Z 432.748,A -85,B 0,C 180,E1 18063.609,E2 18063.609} C_VEL
LIN {X 0,Y 373.69,Z 428.02,A -85,B 0,C 180,E1 18062.331,E2 18062.331} C_VEL
LIN {X 0,Y 371.669,Z 423.972,A -85,B 0,C 180,E1 18061.211,E2 18061.211} C_VEL
LIN {X 0,Y 369.878,Z 420.403,A -85,B 0,C 180,E1 18060.17,E2 18060.17} C_VEL
LIN {X 0,Y 369.746,Z 419.753,A -85,B 0,C 180,E1 18059.8,E2 18059.8} C_VEL
LIN {X 0,Y 369.736,Z 419.66,A -85,B 0,C 180,E1 18055.769,E2 18055.769} C_VEL
LIN {X 0,Y 369.741,Z 419.657,A -85,B 0,C 180,E1 18051.649,E2 18051.649} C_VEL
LIN {X 0,Y 369.74,Z 419.66,A -85,B 0,C 180,E1 18047.583,E2 18047.583} C_VEL
LIN {X 0,Y 369.741,Z 419.67,A -85,B 0,C 180,E1 18043.384,E2 18043.384} C_VEL
LIN {X 0,Y 369.748,Z 419.679,A -85,B 0,C 180,E1 18039.256,E2 18039.256} C_VEL
LIN {X 0,Y 369.74,Z 419.664,A -85,B 0,C 180,E1 18035.17,E2 18035.17} C_VEL
LIN {X 0,Y 369.744,Z 419.649,A -85,B 0,C 180,E1 18030.99,E2 18030.99} C_VEL
LIN {X 0,Y 369.742,Z 419.653,A -85,B 0,C 180,E1 18026.822,E2 18026.822} C_VEL
LIN {X 0,Y 369.745,Z 419.675,A -85,B 0,C 180,E1 18022.582,E2 18022.582} C_VEL
LIN {X 0,Y 369.741,Z 419.665,A -85,B 0,C 180,E1 18018.445,E2 18018.445} C_VEL
LIN {X 0,Y 369.741,Z 419.648,A -85,B 0,C 180,E1 18014.246,E2 18014.246} C_VEL
LIN {X 0,Y 369.741,Z 419.661,A -85,B 0,C 180,E1 18010.124,E2 18010.124} C_VEL
LIN {X 0,Y 369.747,Z 419.679,A -85,B 0,C 180,E1 18006.054,E2 18006.054} C_VEL
LIN {X 0,Y 369.74,Z 419.658,A -85,B 0,C 180,E1 18001.86,E2 18001.86} C_VEL
LIN {X 0,Y 369.739,Z 419.65,A -85,B 0,C 180,E1 17997.831,E2 17997.831} C_VEL
LIN {X 0,Y 369.743,Z 419.655,A -85,B 0,C 180,E1 17993.635,E2 17993.635} C_VEL
LIN {X 0,Y 369.741,Z 419.673,A -85,B 0,C 180,E1 17989.562,E2 17989.562} C_VEL
LIN {X 0,Y 369.751,Z 419.679,A -85,B 0,C 180,E1 17985.435,E2 17985.435} C_VEL
LIN {X 0,Y 369.745,Z 419.68,A -85,B 0,C 180,E1 17981.229,E2 17981.229} C_VEL
LIN {X 0,Y 369.75,Z 419.679,A -85,B 0,C 180,E1 17977.084,E2 17977.084} C_VEL
LIN {X 0,Y 369.763,Z 419.816,A -85,B 0,C 180,E1 17972.982,E2 17972.982} C_VEL
LIN {X 0,Y 369.925,Z 420.626,A -85,B 0,C 180,E1 17972.646,E2 17972.646} C_VEL
LIN {X 0,Y 371.93,Z 424.268,A -85,B 0,C 180,E1 17971.587,E2 17971.587} C_VEL
LIN {X 0,Y 375.57,Z 430.975,A -85,B 0,C 180,E1 17969.791,E2 17969.791} C_VEL
LIN {X 0,Y 378.102,Z 435.574,A -85,B 0,C 180,E1 17968.605,E2 17968.605} C_VEL
LIN {X 0,Y 384.689,Z 447.996,A -85,B 0,C 180,E1 17965.667,E2 17965.667} C_VEL
LIN {X 0,Y 388.459,Z 455.283,A -85,B 0,C 180,E1 17964.158,E2 17964.158} C_VEL
LIN {X 0,Y 401.094,Z 473.923,A -85,B 0,C 180,E1 17961.564,E2 17961.564} C_VEL
LIN {X 0,Y 413.193,Z 493.251,A -85,B 0,C 180,E1 17959.274,E2 17959.274} C_VEL
LIN {X 0,Y 417.368,Z 500.8,A -85,B 0,C 180,E1 17958.51,E2 17958.51} C_VEL
LIN {X 0,Y 409.303,Z 718.077,A -85,B 0,C 180,E1 17954.443,E2 17954.443} C_VEL
LIN {X 0,Y 407.689,Z 757.743,A -85,B 0,C 180,E1 17953.667,E2 17953.667} C_VEL
LIN {X 0,Y 405.749,Z 779.681,A -85,B 0,C 180,E1 17953.031,E2 17953.031} C_VEL
LIN {X 0,Y 403.26,Z 800.73,A -85,B 0,C 180,E1 17952.173,E2 17952.173} C_VEL
LIN {X 0,Y 400.307,Z 821.595,A -85,B 0,C 180,E1 17951.067,E2 17951.067} C_VEL
LIN {X 0,Y 397.058,Z 841.159,A -85,B 0,C 180,E1 17949.766,E2 17949.766} C_VEL
LIN {X 0,Y 393.309,Z 860.879,A -85,B 0,C 180,E1 17948.154,E2 17948.154} C_VEL
LIN {X 0,Y 389.32,Z 880.518,A -85,B 0,C 180,E1 17946.209,E2 17946.209} C_VEL
LIN {X 0,Y 385.691,Z 897.494,A -85,B 0,C 180,E1 17944.212,E2 17944.212} C_VEL
LIN {X 0,Y 381.921,Z 914.423,A -85,B 0,C 180,E1 17941.841,E2 17941.841} C_VEL
LIN {X 0,Y 378.479,Z 929.965,A -85,B 0,C 180,E1 17939.26,E2 17939.26} C_VEL
LIN {X 0,Y 375.393,Z 944.49,A -85,B 0,C 180,E1 17936.413,E2 17936.413} C_VEL
LIN {X 0,Y 372.937,Z 957,A -85,B 0,C 180,E1 17933.522,E2 17933.522} C_VEL
LIN {X 0,Y 370.933,Z 968.39,A -85,B 0,C 180,E1 17930.351,E2 17930.351} C_VEL
LIN {X 0,Y 369.558,Z 977.9,A -85,B 0,C 180,E1 17927.155,E2 17927.155} C_VEL
LIN {X 0,Y 368.707,Z 985.659,A -85,B 0,C 180,E1 17923.969,E2 17923.969} C_VEL
LIN {X 0,Y 368.274,Z 991.625,A -85,B 0,C 180,E1 17920.8,E2 17920.8} C_VEL
LIN {X 0,Y 368.089,Z 996.23,A -85,B 0,C 180,E1 17917.493,E2 17917.493} C_VEL
LIN {X 0,Y 368.086,Z 998.825,A -85,B 0,C 180,E1 17914.677,E2 17914.677} C_VEL
LIN {X 0,Y 368.121,Z 1000.316,A -85,B 0,C 180,E1 17911.404,E2 17911.404} C_VEL
LIN {X 0,Y 368.125,Z 1000.285,A -85,B 0,C 180,E1 17908.603,E2 17908.603} C_VEL
LIN {X 0,Y 368.093,Z 998.722,A -85,B 0,C 180,E1 17905.329,E2 17905.329} C_VEL
LIN {X 0,Y 368.101,Z 996.037,A -85,B 0,C 180,E1 17902.493,E2 17902.493} C_VEL
LIN {X 0,Y 368.284,Z 991.378,A -85,B 0,C 180,E1 17899.207,E2 17899.207} C_VEL
LIN {X 0,Y 368.709,Z 985.319,A -85,B 0,C 180,E1 17896.038,E2 17896.038} C_VEL
LIN {X 0,Y 369.547,Z 977.459,A -85,B 0,C 180,E1 17892.852,E2 17892.852} C_VEL
LIN {X 0,Y 370.989,Z 967.304,A -85,B 0,C 180,E1 17889.495,E2 17889.495} C_VEL
LIN {X 0,Y 372.903,Z 956.253,A -85,B 0,C 180,E1 17886.457,E2 17886.457} C_VEL
LIN {X 0,Y 375.47,Z 943.002,A -85,B 0,C 180,E1 17883.429,E2 17883.429} C_VEL
LIN {X 0,Y 378.464,Z 928.743,A -85,B 0,C 180,E1 17880.67,E2 17880.67} C_VEL
LIN {X 0,Y 381.913,Z 912.989,A -85,B 0,C 180,E1 17878.078,E2 17878.078} C_VEL
LIN {X 0,Y 385.732,Z 895.812,A -85,B 0,C 180,E1 17875.687,E2 17875.687} C_VEL
LIN {X 0,Y 389.482,Z 878.203,A -85,B 0,C 180,E1 17873.634,E2 17873.634} C_VEL
LIN {X 0,Y 393.378,Z 859.055,A -85,B 0,C 180,E1 17871.756,E2 17871.756} C_VEL
LIN {X 0,Y 397.091,Z 839.581,A -85,B 0,C 180,E1 17870.172,E2 17870.172} C_VEL
LIN {X 0,Y 400.396,Z 819.854,A -85,B 0,C 180,E1 17868.864,E2 17868.864} C_VEL
LIN {X 0,Y 403.412,Z 798.896,A -85,B 0,C 180,E1 17867.757,E2 17867.757} C_VEL
LIN {X 0,Y 406.031,Z 777.084,A -85,B 0,C 180,E1 17866.882,E2 17866.882} C_VEL
LIN {X 0,Y 407.977,Z 755.057,A -85,B 0,C 180,E1 17866.251,E2 17866.251} C_VEL
LIN {X 0,Y 411.036,Z 674.755,A -85,B 0,C 180,E1 17864.721,E2 17864.721} C_VEL
LIN {X 0,Y 417.945,Z 500.12,A -85,B 0,C 180,E1 17861.396,E2 17861.396} C_VEL
LIN {X 0,Y 408.349,Z 483.329,A -85,B 0,C 180,E1 17859.426,E2 17859.426} C_VEL
LIN {X 0,Y 397.681,Z 466.781,A -85,B 0,C 180,E1 17857.024,E2 17857.024} C_VEL
LIN {X 0,Y 388.8,Z 453.983,A -85,B 0,C 180,E1 17854.723,E2 17854.723} C_VEL
LIN {X 0,Y 383.829,Z 444.659,A -85,B 0,C 180,E1 17852.1,E2 17852.1} C_VEL
LIN {X 0,Y 381.218,Z 439.919,A -85,B 0,C 180,E1 17850.585,E2 17850.585} C_VEL
LIN {X 0,Y 378.825,Z 435.457,A -85,B 0,C 180,E1 17849.054,E2 17849.054} C_VEL
LIN {X 0,Y 376.703,Z 432.035,A -85,B 0,C 180,E1 17847.677,E2 17847.677} C_VEL
LIN {X 0,Y 375.929,Z 430.414,A -85,B 0,C 180,E1 17847.052,E2 17847.052} C_VEL
LIN {X 0,Y 373.583,Z 426.867,A -85,B 0,C 180,E1 17845.354,E2 17845.354} C_VEL
LIN {X 0,Y 372.766,Z 425.122,A -85,B 0,C 180,E1 17844.566,E2 17844.566} C_VEL
LIN {X 0,Y 370.197,Z 421.661,A -85,B 0,C 180,E1 17842.384,E2 17842.384} C_VEL
LIN {X 0,Y 369.727,Z 419.853,A -85,B 0,C 180,E1 17841.246,E2 17841.246} C_VEL
LIN {X 0,Y 369.704,Z 419.671,A -85,B 0,C 180,E1 17837.307,E2 17837.307} C_VEL
LIN {X 0,Y 369.706,Z 419.684,A -85,B 0,C 180,E1 17833.214,E2 17833.214} C_VEL
LIN {X 0,Y 369.713,Z 419.673,A -85,B 0,C 180,E1 17829.181,E2 17829.181} C_VEL
LIN {X 0,Y 369.725,Z 419.667,A -85,B 0,C 180,E1 17825.275,E2 17825.275} C_VEL
LIN {X 0,Y 369.757,Z 419.828,A -85,B 0,C 180,E1 17821.084,E2 17821.084} C_VEL
LIN {X 0,Y 370.033,Z 421.192,A -85,B 0,C 180,E1 17820.154,E2 17820.154} C_VEL
LIN {X 0,Y 372.705,Z 425.059,A -85,B 0,C 180,E1 17817.693,E2 17817.693} C_VEL
LIN {X 0,Y 375.088,Z 429.589,A -85,B 0,C 180,E1 17815.566,E2 17815.566} C_VEL
LIN {X 0,Y 376.138,Z 431.155,A -85,B 0,C 180,E1 17814.814,E2 17814.814} C_VEL
LIN {X 0,Y 378.145,Z 434.831,A -85,B 0,C 180,E1 17813.319,E2 17813.319} C_VEL
LIN {X 0,Y 381.395,Z 440.939,A -85,B 0,C 180,E1 17811.102,E2 17811.102} C_VEL
LIN {X 0,Y 384.117,Z 446.45,A -85,B 0,C 180,E1 17809.349,E2 17809.349} C_VEL
LIN {X 0,Y 387.644,Z 453.339,A -85,B 0,C 180,E1 17807.335,E2 17807.335} C_VEL
LIN {X 0,Y 397.356,Z 467.413,A -85,B 0,C 180,E1 17804.773,E2 17804.773} C_VEL
LIN {X 0,Y 406.349,Z 481.346,A -85,B 0,C 180,E1 17802.674,E2 17802.674} C_VEL
LIN {X 0,Y 416.032,Z 498.003,A -85,B 0,C 180,E1 17800.605,E2 17800.605} C_VEL
LIN {X 0,Y 405.377,Z 724.01,A -85,B 0,C 180,E1 17796.1,E2 17796.1} C_VEL
LIN {X 0,Y 403.658,Z 744.823,A -85,B 0,C 180,E1 17795.436,E2 17795.436} C_VEL
LIN {X 0,Y 401.425,Z 764.587,A -85,B 0,C 180,E1 17794.562,E2 17794.562} C_VEL
LIN {X 0,Y 398.596,Z 784.877,A -85,B 0,C 180,E1 17793.387,E2 17793.387} C_VEL
LIN {X 0,Y 395.451,Z 803.788,A -85,B 0,C 180,E1 17792.01,E2 17792.01} C_VEL
LIN {X 0,Y 392.05,Z 821.686,A -85,B 0,C 180,E1 17790.41,E2 17790.41} C_VEL
LIN {X 0,Y 388.365,Z 839.28,A -85,B 0,C 180,E1 17788.491,E2 17788.491} C_VEL
LIN {X 0,Y 384.586,Z 855.913,A -85,B 0,C 180,E1 17786.291,E2 17786.291} C_VEL
LIN {X 0,Y 381.199,Z 870.198,A -85,B 0,C 180,E1 17784.017,E2 17784.017} C_VEL
LIN {X 0,Y 378.046,Z 883.374,A -85,B 0,C 180,E1 17781.516,E2 17781.516} C_VEL
LIN {X 0,Y 375.167,Z 895.62,A -85,B 0,C 180,E1 17778.719,E2 17778.719} C_VEL
LIN {X 0,Y 372.914,Z 905.719,A -85,B 0,C 180,E1 17775.929,E2 17775.929} C_VEL
LIN {X 0,Y 371.085,Z 914.717,A -85,B 0,C 180,E1 17772.871,E2 17772.871} C_VEL
LIN {X 0,Y 369.759,Z 922.127,A -85,B 0,C 180,E1 17769.649,E2 17769.649} C_VEL
LIN {X 0,Y 368.99,Z 927.428,A -85,B 0,C 180,E1 17766.588,E2 17766.588} C_VEL
LIN {X 0,Y 368.548,Z 931.403,A -85,B 0,C 180,E1 17763.321,E2 17763.321} C_VEL
LIN {X 0,Y 368.353,Z 933.674,A -85,B 0,C 180,E1 17760.138,E2 17760.138} C_VEL
LIN {X 0,Y 368.301,Z 934.392,A -85,B 0,C 180,E1 17757.069,E2 17757.069} C_VEL
LIN {X 0,Y 368.328,Z 933.594,A -85,B 0,C 180,E1 17754.024,E2 17754.024} C_VEL
LIN {X 0,Y 368.487,Z 931.244,A -85,B 0,C 180,E1 17750.817,E2 17750.817} C_VEL
LIN {X 0,Y 368.865,Z 927.369,A -85,B 0,C 180,E1 17747.669,E2 17747.669} C_VEL
LIN {X 0,Y 369.558,Z 921.949,A -85,B 0,C 180,E1 17744.569,E2 17744.569} C_VEL
LIN {X 0,Y 370.638,Z 915.123,A -85,B 0,C 180,E1 17741.626,E2 17741.626} C_VEL
LIN {X 0,Y 370.191,Z 912.363,A -85,B 0,C 180,E1 17740.506,E2 17740.506} C_VEL
LIN {X 0,Y 365.831,Z 904.607,A -85,B 0,C 180,E1 17737.502,E2 17737.502} C_VEL
LIN {X 0,Y 365.782,Z 901.545,A -85,B 0,C 180,E1 17736.571,E2 17736.571} C_VEL
LIN {X 0,Y 368.458,Z 889.794,A -85,B 0,C 180,E1 17733.575,E2 17733.575} C_VEL
LIN {X 0,Y 371.45,Z 877.191,A -85,B 0,C 180,E1 17730.922,E2 17730.922} C_VEL
LIN {X 0,Y 374.756,Z 863.251,A -85,B 0,C 180,E1 17728.468,E2 17728.468} C_VEL
LIN {X 0,Y 378.448,Z 847.281,A -85,B 0,C 180,E1 17726.134,E2 17726.134} C_VEL
LIN {X 0,Y 382.156,Z 830.126,A -85,B 0,C 180,E1 17724.065,E2 17724.065} C_VEL
LIN {X 0,Y 385.624,Z 812.644,A -85,B 0,C 180,E1 17722.323,E2 17722.323} C_VEL
LIN {X 0,Y 388.972,Z 793.783,A -85,B 0,C 180,E1 17720.782,E2 17720.782} C_VEL
LIN {X 0,Y 391.992,Z 774.037,A -85,B 0,C 180,E1 17719.489,E2 17719.489} C_VEL
LIN {X 0,Y 394.487,Z 754.136,A -85,B 0,C 180,E1 17718.47,E2 17718.47} C_VEL
LIN {X 0,Y 396.508,Z 733.15,A -85,B 0,C 180,E1 17717.671,E2 17717.671} C_VEL
LIN {X 0,Y 397.902,Z 710.963,A -85,B 0,C 180,E1 17717.109,E2 17717.109} C_VEL
LIN {X 0,Y 406.884,Z 499.156,A -85,B 0,C 180,E1 17712.994,E2 17712.994} C_VEL
LIN {X 0,Y 396.114,Z 480.753,A -85,B 0,C 180,E1 17710.908,E2 17710.908} C_VEL
LIN {X 0,Y 384.989,Z 463.542,A -85,B 0,C 180,E1 17708.602,E2 17708.602} C_VEL
LIN {X 0,Y 377.611,Z 452.63,A -85,B 0,C 180,E1 17706.926,E2 17706.926} C_VEL
LIN {X 0,Y 372.606,Z 442.229,A -85,B 0,C 180,E1 17704.374,E2 17704.374} C_VEL
LIN {X 0,Y 368.301,Z 433.729,A -85,B 0,C 180,E1 17702.089,E2 17702.089} C_VEL
LIN {X 0,Y 366.158,Z 429.564,A -85,B 0,C 180,E1 17700.906,E2 17700.906} C_VEL
LIN {X 0,Y 363.705,Z 424.936,A -85,B 0,C 180,E1 17699.525,E2 17699.525} C_VEL
LIN {X 0,Y 361.903,Z 421.244,A -85,B 0,C 180,E1 17698.38,E2 17698.38} C_VEL
LIN {X 0,Y 361.798,Z 420.66,A -85,B 0,C 180,E1 17697.743,E2 17697.743} C_VEL
LIN {X 0,Y 361.798,Z 420.662,A -85,B 0,C 180,E1 17693.534,E2 17693.534} C_VEL
LIN {X 0,Y 361.801,Z 420.657,A -85,B 0,C 180,E1 17689.463,E2 17689.463} C_VEL
LIN {X 0,Y 361.796,Z 420.65,A -85,B 0,C 180,E1 17685.256,E2 17685.256} C_VEL
LIN {X 0,Y 361.798,Z 420.643,A -85,B 0,C 180,E1 17681.019,E2 17681.019} C_VEL
LIN {X 0,Y 361.795,Z 420.639,A -85,B 0,C 180,E1 17676.849,E2 17676.849} C_VEL
LIN {X 0,Y 361.8,Z 420.653,A -85,B 0,C 180,E1 17672.797,E2 17672.797} C_VEL
LIN {X 0,Y 361.804,Z 420.667,A -85,B 0,C 180,E1 17668.561,E2 17668.561} C_VEL
LIN {X 0,Y 361.798,Z 420.648,A -85,B 0,C 180,E1 17664.317,E2 17664.317} C_VEL
LIN {X 0,Y 361.799,Z 420.634,A -85,B 0,C 180,E1 17660.21,E2 17660.21} C_VEL
LIN {X 0,Y 361.799,Z 420.654,A -85,B 0,C 180,E1 17656.043,E2 17656.043} C_VEL
LIN {X 0,Y 361.803,Z 420.668,A -85,B 0,C 180,E1 17651.801,E2 17651.801} C_VEL
LIN {X 0,Y 361.802,Z 420.644,A -85,B 0,C 180,E1 17647.623,E2 17647.623} C_VEL
LIN {X 0,Y 361.797,Z 420.635,A -85,B 0,C 180,E1 17643.486,E2 17643.486} C_VEL
LIN {X 0,Y 361.802,Z 420.652,A -85,B 0,C 180,E1 17639.367,E2 17639.367} C_VEL
LIN {X 0,Y 361.803,Z 420.667,A -85,B 0,C 180,E1 17635.086,E2 17635.086} C_VEL
LIN {X 0,Y 361.805,Z 420.659,A -85,B 0,C 180,E1 17630.937,E2 17630.937} C_VEL
LIN {X 0,Y 361.806,Z 420.649,A -85,B 0,C 180,E1 17626.74,E2 17626.74} C_VEL
LIN {X 0,Y 361.804,Z 420.645,A -85,B 0,C 180,E1 17622.635,E2 17622.635} C_VEL
LIN {X 0,Y 361.809,Z 420.646,A -85,B 0,C 180,E1 17618.436,E2 17618.436} C_VEL
LIN {X 0,Y 361.836,Z 420.878,A -85,B 0,C 180,E1 17614.684,E2 17614.684} C_VEL
LIN {X 0,Y 363.168,Z 424.24,A -85,B 0,C 180,E1 17613.689,E2 17613.689} C_VEL
LIN {X 0,Y 364.771,Z 426.491,A -85,B 0,C 180,E1 17612.935,E2 17612.935} C_VEL
LIN {X 0,Y 366.802,Z 430.214,A -85,B 0,C 180,E1 17611.864,E2 17611.864} C_VEL
LIN {X 0,Y 370.693,Z 437.508,A -85,B 0,C 180,E1 17609.889,E2 17609.889} C_VEL
LIN {X 0,Y 374.881,Z 445.049,A -85,B 0,C 180,E1 17607.944,E2 17607.944} C_VEL
LIN {X 0,Y 380.049,Z 455.077,A -85,B 0,C 180,E1 17605.668,E2 17605.668} C_VEL
LIN {X 0,Y 392.102,Z 472.456,A -85,B 0,C 180,E1 17603.047,E2 17603.047} C_VEL
LIN {X 0,Y 404.321,Z 491.554,A -85,B 0,C 180,E1 17600.609,E2 17600.609} C_VEL
LIN {X 0,Y 411.577,Z 504.106,A -85,B 0,C 180,E1 17599.233,E2 17599.233} C_VEL
LIN {X 0,Y 403.021,Z 724.725,A -85,B 0,C 180,E1 17595.061,E2 17595.061} C_VEL
LIN {X 0,Y 401.51,Z 758.356,A -85,B 0,C 180,E1 17594.382,E2 17594.382} C_VEL
LIN {X 0,Y 399.479,Z 780.332,A -85,B 0,C 180,E1 17593.732,E2 17593.732} C_VEL
LIN {X 0,Y 396.831,Z 801.554,A -85,B 0,C 180,E1 17592.845,E2 17592.845} C_VEL
LIN {X 0,Y 393.674,Z 822.646,A -85,B 0,C 180,E1 17591.695,E2 17591.695} C_VEL
LIN {X 0,Y 390.358,Z 841.821,A -85,B 0,C 180,E1 17590.396,E2 17590.396} C_VEL
LIN {X 0,Y 386.379,Z 861.789,A -85,B 0,C 180,E1 17588.726,E2 17588.726} C_VEL
LIN {X 0,Y 382.467,Z 880.094,A -85,B 0,C 180,E1 17586.875,E2 17586.875} C_VEL
LIN {X 0,Y 378.52,Z 897.669,A -85,B 0,C 180,E1 17584.765,E2 17584.765} C_VEL
LIN {X 0,Y 374.706,Z 913.98,A -85,B 0,C 180,E1 17582.438,E2 17582.438} C_VEL
LIN {X 0,Y 371.11,Z 929.434,A -85,B 0,C 180,E1 17579.826,E2 17579.826} C_VEL
LIN {X 0,Y 367.857,Z 943.916,A -85,B 0,C 180,E1 17576.936,E2 17576.936} C_VEL
LIN {X 0,Y 365.192,Z 956.713,A -85,B 0,C 180,E1 17573.907,E2 17573.907} C_VEL
LIN {X 0,Y 363.156,Z 967.6,A -85,B 0,C 180,E1 17570.807,E2 17570.807} C_VEL
LIN {X 0,Y 361.654,Z 977.292,A -85,B 0,C 180,E1 17567.483,E2 17567.483} C_VEL
LIN {X 0,Y 360.763,Z 984.924,A -85,B 0,C 180,E1 17564.283,E2 17564.283} C_VEL
LIN {X 0,Y 360.302,Z 990.898,A -85,B 0,C 180,E1 17561.042,E2 17561.042} C_VEL
LIN {X 0,Y 360.11,Z 995.578,A -85,B 0,C 180,E1 17557.6,E2 17557.6} C_VEL
LIN {X 0,Y 360.112,Z 998.237,A -85,B 0,C 180,E1 17554.612,E2 17554.612} C_VEL
LIN {X 0,Y 360.154,Z 999.628,A -85,B 0,C 180,E1 17551.276,E2 17551.276} C_VEL
LIN {X 0,Y 360.153,Z 999.54,A -85,B 0,C 180,E1 17548.413,E2 17548.413} C_VEL
LIN {X 0,Y 360.116,Z 997.997,A -85,B 0,C 180,E1 17545.226,E2 17545.226} C_VEL
LIN {X 0,Y 360.123,Z 995.321,A -85,B 0,C 180,E1 17542.345,E2 17542.345} C_VEL
LIN {X 0,Y 360.311,Z 990.623,A -85,B 0,C 180,E1 17538.965,E2 17538.965} C_VEL
LIN {X 0,Y 360.765,Z 984.554,A -85,B 0,C 180,E1 17535.724,E2 17535.724} C_VEL
LIN {X 0,Y 361.662,Z 976.679,A -85,B 0,C 180,E1 17532.466,E2 17532.466} C_VEL
LIN {X 0,Y 363.215,Z 966.498,A -85,B 0,C 180,E1 17529.035,E2 17529.035} C_VEL
LIN {X 0,Y 365.261,Z 955.432,A -85,B 0,C 180,E1 17525.933,E2 17525.933} C_VEL
LIN {X 0,Y 367.996,Z 942.174,A -85,B 0,C 180,E1 17522.846,E2 17522.846} C_VEL
LIN {X 0,Y 371.095,Z 928.271,A -85,B 0,C 180,E1 17520.107,E2 17520.107} C_VEL
LIN {X 0,Y 374.721,Z 912.616,A -85,B 0,C 180,E1 17517.476,E2 17517.476} C_VEL
LIN {X 0,Y 378.584,Z 896.091,A -85,B 0,C 180,E1 17515.13,E2 17515.13} C_VEL
LIN {X 0,Y 382.5,Z 878.662,A -85,B 0,C 180,E1 17513.048,E2 17513.048} C_VEL
LIN {X 0,Y 386.717,Z 859.061,A -85,B 0,C 180,E1 17511.082,E2 17511.082} C_VEL
LIN {X 0,Y 390.555,Z 839.949,A -85,B 0,C 180,E1 17509.494,E2 17509.494} C_VEL
LIN {X 0,Y 394.063,Z 819.905,A -85,B 0,C 180,E1 17508.146,E2 17508.146} C_VEL
LIN {X 0,Y 397.29,Z 798.56,A -85,B 0,C 180,E1 17507.004,E2 17507.004} C_VEL
LIN {X 0,Y 400,Z 777.066,A -85,B 0,C 180,E1 17506.13,E2 17506.13} C_VEL
LIN {X 0,Y 402.014,Z 755.305,A -85,B 0,C 180,E1 17505.497,E2 17505.497} C_VEL
LIN {X 0,Y 403.983,Z 708.647,A -85,B 0,C 180,E1 17504.578,E2 17504.578} C_VEL
LIN {X 0,Y 412.424,Z 504.397,A -85,B 0,C 180,E1 17500.659,E2 17500.659} C_VEL
LIN {X 0,Y 412.209,Z 503.13,A -85,B 0,C 180,E1 17500.592,E2 17500.592} C_VEL
LIN {X 0,Y 403.604,Z 488.062,A -85,B 0,C 180,E1 17498.743,E2 17498.743} C_VEL
LIN {X 0,Y 394.213,Z 473.177,A -85,B 0,C 180,E1 17496.541,E2 17496.541} C_VEL
LIN {X 0,Y 384.749,Z 459.71,A -85,B 0,C 180,E1 17494.057,E2 17494.057} C_VEL
LIN {X 0,Y 380.541,Z 453.913,A -85,B 0,C 180,E1 17492.769,E2 17492.769} C_VEL
LIN {X 0,Y 378.374,Z 449.89,A -85,B 0,C 180,E1 17491.548,E2 17491.548} C_VEL
LIN {X 0,Y 376.391,Z 446.078,A -85,B 0,C 180,E1 17490.312,E2 17490.312} C_VEL
LIN {X 0,Y 373.973,Z 441.625,A -85,B 0,C 180,E1 17488.734,E2 17488.734} C_VEL
LIN {X 0,Y 371.863,Z 437.693,A -85,B 0,C 180,E1 17487.199,E2 17487.199} C_VEL
LIN {X 0,Y 369.004,Z 433.046,A -85,B 0,C 180,E1 17485.005,E2 17485.005} C_VEL
LIN {X 0,Y 368.115,Z 431.494,A -85,B 0,C 180,E1 17484.213,E2 17484.213} C_VEL
LIN {X 0,Y 365.762,Z 427.913,A -85,B 0,C 180,E1 17481.993,E2 17481.993} C_VEL
LIN {X 0,Y 365.063,Z 426.296,A -85,B 0,C 180,E1 17481.026,E2 17481.026} C_VEL
LIN {X 0,Y 361.874,Z 421.385,A -85,B 0,C 180,E1 17475.964,E2 17475.964} C_VEL
LIN {X 0,Y 361.77,Z 420.745,A -85,B 0,C 180,E1 17473.75,E2 17473.75} C_VEL
LIN {X 0,Y 361.78,Z 420.715,A -85,B 0,C 180,E1 17469.545,E2 17469.545} C_VEL
LIN {X 0,Y 361.82,Z 421.118,A -85,B 0,C 180,E1 17466.665,E2 17466.665} C_VEL
LIN {X 0,Y 365.017,Z 426.225,A -85,B 0,C 180,E1 17461.255,E2 17461.255} C_VEL
LIN {X 0,Y 367.601,Z 431.032,A -85,B 0,C 180,E1 17458.285,E2 17458.285} C_VEL
LIN {X 0,Y 368.524,Z 432.254,A -85,B 0,C 180,E1 17457.512,E2 17457.512} C_VEL
LIN {X 0,Y 370.319,Z 435.88,A -85,B 0,C 180,E1 17455.819,E2 17455.819} C_VEL
LIN {X 0,Y 371.356,Z 437.386,A -85,B 0,C 180,E1 17455.057,E2 17455.057} C_VEL
LIN {X 0,Y 373.55,Z 441.369,A -85,B 0,C 180,E1 17453.39,E2 17453.39} C_VEL
LIN {X 0,Y 376.633,Z 447.626,A -85,B 0,C 180,E1 17451.142,E2 17451.142} C_VEL
LIN {X 0,Y 379.359,Z 453.124,A -85,B 0,C 180,E1 17449.368,E2 17449.368} C_VEL
